LIN {X -195.246,Y +1107.046,Z +0.000,A -20.000,E1 +44.515,E3 +167624.420,E4 +0.000} C_DIS
LIN {X -198.051,Y +1092.368,Z +0.000,A -20.000,E1 +47.947,E3 +167640.946,E4 +0.000} C_DIS
LIN {X -198.143,Y +1081.370,Z +0.000,A -19.806,E1 +49.153,E3 +167652.807,E4 +0.000} C_DIS
LIN {X -197.177,Y +1073.569,Z +0.000,A -17.356,E1 +49.162,E3 +167661.391,E4 +0.000} C_DIS
LIN {X -195.448,Y +1066.139,Z +0.000,A -12.154,E1 +48.512,E3 +167669.986,E4 +0.000} C_DIS
LIN {X -193.346,Y +1058.941,Z +0.000,A -7.133,E1 +47.724,E3 +167678.866,E4 +0.000} C_DIS
LIN {X -191.781,Y +1050.839,Z +0.000,A -3.715,E1 +47.274,E3 +167689.199,E4 +0.000} C_DIS
LIN {X -190.795,Y +1039.355,Z +0.000,A -0.983,E1 +46.842,E3 +167703.859,E4 +0.000} C_DIS
LIN {X -190.395,Y +1028.856,Z +0.000,A -0.089,E1 +46.598,E3 +167717.253,E4 +0.000} C_DIS
LIN {X -190.239,Y +1018.851,Z +0.000,A -0.004,E1 +46.529,E3 +167730.021,E4 +0.000} C_DIS
LIN {X -190.161,Y +1004.975,Z +0.000,A +0.000,E1 +46.506,E3 +167747.735,E4 +0.000} C_DIS
LIN {X -190.142,Y +412.853,Z +0.000,A +0.000,E1 +46.501,E3 +168503.941,E4 +0.000} C_DIS
LIN {X -190.147,Y +401.077,Z +0.000,A +0.000,E1 +46.499,E3 +168518.982,E4 +0.000} C_DIS
LIN {X -190.159,Y +390.929,Z +0.000,A +0.000,E1 +46.494,E3 +168531.948,E4 +0.000} C_DIS
LIN {X -190.174,Y +383.973,Z +0.000,A +0.000,E1 +46.484,E3 +168540.841,E4 +0.000} C_DIS
LIN {X -190.200,Y +373.815,Z +0.000,A +0.000,E1 +46.448,E3 +168553.846,E4 +0.000} C_DIS
LIN {X -190.154,Y +361.003,Z +0.000,A +0.000,E1 +46.303,E3 +168570.340,E4 +0.000} C_DIS
LIN {X -189.772,Y +350.660,Z +0.000,A +0.049,E1 +45.996,E3 +168583.879,E4 +0.000} C_DIS
LIN {X -189.325,Y +346.917,Z +0.000,A +0.243,E1 +45.771,E3 +168588.948,E4 +0.000} C_DIS
LIN {X -188.196,Y +342.754,Z +0.000,A +1.966,E1 +45.249,E3 +168594.956,E4 +0.000} C_DIS
LIN {X -185.199,Y +337.023,Z +0.000,A +6.630,E1 +43.793,E3 +168604.330,E4 +0.000} C_DIS
LIN {X -181.141,Y +331.596,Z +0.000,A +12.274,E1 +41.569,E3 +168614.890,E4 +0.000} C_DIS
LIN {X -176.762,Y +326.804,Z +0.000,A +17.560,E1 +38.898,E3 +168626.314,E4 +0.000} C_DIS
LIN {X -172.184,Y +322.578,Z +0.000,A +19.859,E1 +36.197,E3 +168639.044,E4 +0.000} C_DIS
LIN {X -165.998,Y +317.874,Z +0.000,A +20.000,E1 +32.027,E3 +168658.802,E4 +0.000} C_DIS
LIN {X -160.137,Y +314.334,Z +0.000,A +20.000,E1 +26.368,E3 +168683.171,E4 +0.000} C_DIS
LIN {X -155.624,Y +312.245,Z +0.000,A +20.000,E1 +19.506,E3 +168711.847,E4 +0.000} C_DIS
LIN {X -153.557,Y +311.879,Z +0.000,A +20.000,E1 +11.113,E3 +168747.602,E4 +0.000} C_DIS
LIN {X -155.320,Y +313.348,Z +0.000,A +20.000,E1 +3.401,E3 +168780.786,E4 +0.000} C_DIS
LIN {X -160.005,Y +315.804,Z +0.000,A +20.000,E1 -4.720,E3 +168811.164,E4 +0.000} C_DIS
LIN {X -164.504,Y +318.255,Z +0.000,A +20.000,E1 -10.663,E3 +168830.533,E4 +0.000} C_DIS
LIN {X -170.340,Y +322.684,Z +0.000,A +20.000,E1 -17.457,E3 +168850.565,E4 +0.000} C_DIS
LIN {X -175.568,Y +329.106,Z +0.000,A +20.000,E1 -24.747,E3 +168867.799,E4 +0.000} C_DIS
LIN {X -184.074,Y +340.065,Z +0.000,A +20.000,E1 -33.664,E3 +168890.739,E4 +0.000} C_DIS
LIN {X -190.779,Y +351.388,Z +0.000,A +20.000,E1 -40.083,E3 +168908.517,E4 +0.000} C_DIS
LIN {X -195.254,Y +362.955,Z +0.000,A +20.000,E1 -44.515,E3 +168923.270,E4 +0.000} C_DIS
LIN {X -197.754,Y +374.780,Z +0.000,A +20.000,E1 -47.450,E3 +168936.692,E4 +0.000} C_DIS
LIN {X -198.310,Y +383.215,Z +0.000,A +19.956,E1 -48.698,E3 +168945.816,E4 +0.000} C_DIS
LIN {X -197.912,Y +391.275,Z +0.000,A +18.601,E1 -49.158,E3 +168954.534,E4 +0.000} C_DIS
LIN {X -196.679,Y +398.944,Z +0.000,A +13.989,E1 -48.784,E3 +168963.088,E4 +0.000} C_DIS
LIN {X -194.742,Y +406.288,Z +0.000,A +8.476,E1 -48.001,E3 +168971.771,E4 +0.000} C_DIS
LIN {X -192.748,Y +413.472,Z +0.000,A +3.905,E1 -47.267,E3 +168980.781,E4 +0.000} C_DIS
LIN {X -191.781,Y +419.162,Z +0.000,A +1.739,E1 -46.975,E3 +168988.049,E4 +0.000} C_DIS
LIN {X -190.795,Y +430.646,Z +0.000,A +0.152,E1 -46.707,E3 +169002.710,E4 +0.000} C_DIS
LIN {X -190.395,Y +441.145,Z +0.000,A +0.001,E1 -46.583,E3 +169016.103,E4 +0.000} C_DIS
LIN {X -190.239,Y +451.150,Z +0.000,A -0.000,E1 -46.528,E3 +169028.871,E4 +0.000} C_DIS
LIN {X -190.161,Y +465.026,Z +0.000,A -0.000,E1 -46.506,E3 +169046.586,E4 +0.000} C_DIS
LIN {X -190.142,Y +1057.148,Z +0.000,A -0.000,E1 -46.500,E3 +169802.792,E4 +0.000} C_DIS
LIN {X -190.147,Y +1068.924,Z +0.000,A -0.000,E1 -46.499,E3 +169817.833,E4 +0.000} C_DIS
LIN {X -190.159,Y +1079.072,Z +0.000,A -0.000,E1 -46.493,E3 +169830.798,E4 +0.000} C_DIS
LIN {X -190.174,Y +1086.028,Z +0.000,A -0.000,E1 -46.483,E3 +169839.692,E4 +0.000} C_DIS
LIN {X -190.200,Y +1096.186,Z +0.000,A -0.000,E1 -46.448,E3 +169852.696,E4 +0.000} C_DIS
LIN {X -190.154,Y +1108.998,Z +0.000,A -0.054,E1 -46.295,E3 +169869.191,E4 +0.000} C_DIS
LIN {X -189.772,Y +1119.341,Z +0.000,A -0.752,E1 -45.902,E3 +169882.729,E4 +0.000} C_DIS
LIN {X -189.097,Y +1124.276,Z +0.000,A -2.508,E1 -45.397,E3 +169889.461,E4 +0.000} C_DIS
LIN {X -187.410,Y +1129.069,Z +0.000,A -5.304,E1 -44.585,E3 +169896.634,E4 +0.000} C_DIS
LIN {X -183.899,Y +1134.873,Z +0.000,A -10.372,E1 -42.805,E3 +169906.640,E4 +0.000} C_DIS
LIN {X -179.711,Y +1140.065,Z +0.000,A -15.940,E1 -40.393,E3 +169917.426,E4 +0.000} C_DIS
LIN {X -176.763,Y +1143.197,Z +0.000,A -18.748,E1 -38.674,E3 +169925.164,E4 +0.000} C_DIS
LIN {X -172.185,Y +1147.423,Z +0.000,A -19.971,E1 -36.175,E3 +169937.894,E4 +0.000} C_DIS
LIN {X -165.999,Y +1152.127,Z +0.000,A -20.000,E1 -32.027,E3 +169957.652,E4 +0.000} C_DIS
LIN {X -160.138,Y +1155.667,Z +0.000,A -20.000,E1 -26.368,E3 +169982.022,E4 +0.000} C_DIS
LIN {X -155.625,Y +1157.756,Z +0.000,A -20.000,E1 -19.505,E3 +170010.698,E4 +0.000} C_DIS
LIN {X -153.552,Y +1158.113,Z +0.000,A -20.000,E1 -11.113,E3 +170046.449,E4 +0.000} C_DIS
LIN {X -156.311,Y +1155.540,Z +0.000,A -20.000,E1 -0.839,E3 +170089.809,E4 +0.000} C_DIS
LIN {X -161.281,Y +1151.851,Z +0.000,A -20.000,E1 +7.737,E3 +170119.708,E4 +0.000} C_DIS
LIN {X -167.493,Y +1147.157,Z +0.000,A -20.000,E1 +16.195,E3 +170144.147,E4 +0.000} C_DIS
LIN {X -173.235,Y +1142.221,Z +0.000,A -20.000,E1 +22.930,E3 +170161.449,E4 +0.000} C_DIS
LIN {X -181.123,Y +1133.734,Z +0.000,A -20.000,E1 +30.868,E3 +170182.205,E4 +0.000} C_DIS
LIN {X -189.654,Y +1120.856,Z +0.000,A -20.000,E1 +39.018,E3 +170204.219,E4 +0.000} C_DIS
LIN {X -195.246,Y +1107.046,Z +0.000,A -20.000,E1 +44.515,E3 +170222.121,E4 +0.000} C_DIS
LIN {X -198.051,Y +1092.368,Z +0.000,A -20.000,E1 +47.947,E3 +170238.647,E4 +0.000} C_DIS
LIN {X -198.143,Y +1081.370,Z +0.000,A -19.806,E1 +49.153,E3 +170250.508,E4 +0.000} C_DIS
LIN {X -197.177,Y +1073.569,Z +0.000,A -17.356,E1 +49.162,E3 +170259.092,E4 +0.000} C_DIS
LIN {X -195.448,Y +1066.139,Z +0.000,A -12.154,E1 +48.512,E3 +170267.687,E4 +0.000} C_DIS
LIN {X -193.346,Y +1058.941,Z +0.000,A -7.133,E1 +47.724,E3 +170276.567,E4 +0.000} C_DIS
LIN {X -191.781,Y +1050.839,Z +0.000,A -3.715,E1 +47.274,E3 +170286.900,E4 +0.000} C_DIS
LIN {X -190.795,Y +1039.355,Z +0.000,A -0.983,E1 +46.842,E3 +170301.560,E4 +0.000} C_DIS
LIN {X -190.395,Y +1028.856,Z +0.000,A -0.089,E1 +46.598,E3 +170314.954,E4 +0.000} C_DIS
LIN {X -190.239,Y +1018.851,Z +0.000,A -0.004,E1 +46.529,E3 +170327.722,E4 +0.000} C_DIS
LIN {X -190.161,Y +1004.975,Z +0.000,A +0.000,E1 +46.506,E3 +170345.436,E4 +0.000} C_DIS
LIN {X -190.142,Y +412.853,Z +0.000,A +0.000,E1 +46.501,E3 +171101.642,E4 +0.000} C_DIS
LIN {X -190.147,Y +401.077,Z +0.000,A +0.000,E1 +46.499,E3 +171116.683,E4 +0.000} C_DIS
LIN {X -190.159,Y +390.929,Z +0.000,A +0.000,E1 +46.494,E3 +171129.649,E4 +0.000} C_DIS
LIN {X -190.174,Y +383.973,Z +0.000,A +0.000,E1 +46.484,E3 +171138.542,E4 +0.000} C_DIS
LIN {X -190.200,Y +373.815,Z +0.000,A +0.000,E1 +46.448,E3 +171151.547,E4 +0.000} C_DIS
LIN {X -190.154,Y +361.003,Z +0.000,A +0.000,E1 +46.303,E3 +171168.041,E4 +0.000} C_DIS
LIN {X -189.772,Y +350.660,Z +0.000,A +0.049,E1 +45.996,E3 +171181.580,E4 +0.000} C_DIS
LIN {X -189.325,Y +346.917,Z +0.000,A +0.243,E1 +45.771,E3 +171186.649,E4 +0.000} C_DIS
LIN {X -188.196,Y +342.754,Z +0.000,A +1.966,E1 +45.249,E3 +171192.657,E4 +0.000} C_DIS
LIN {X -185.199,Y +337.023,Z +0.000,A +6.630,E1 +43.793,E3 +171202.031,E4 +0.000} C_DIS
LIN {X -181.141,Y +331.596,Z +0.000,A +12.274,E1 +41.569,E3 +171212.591,E4 +0.000} C_DIS
LIN {X -176.762,Y +326.804,Z +0.000,A +17.560,E1 +38.898,E3 +171224.015,E4 +0.000} C_DIS
LIN {X -172.184,Y +322.578,Z +0.000,A +19.859,E1 +36.197,E3 +171236.745,E4 +0.000} C_DIS
LIN {X -165.998,Y +317.874,Z +0.000,A +20.000,E1 +32.027,E3 +171256.503,E4 +0.000} C_DIS
LIN {X -160.137,Y +314.334,Z +0.000,A +20.000,E1 +26.368,E3 +171280.872,E4 +0.000} C_DIS
LIN {X -155.624,Y +312.245,Z +0.000,A +20.000,E1 +19.506,E3 +171309.548,E4 +0.000} C_DIS
LIN {X -153.557,Y +311.879,Z +0.000,A +20.000,E1 +11.113,E3 +171345.303,E4 +0.000} C_DIS
LIN {X -155.320,Y +313.348,Z +0.000,A +20.000,E1 +3.401,E3 +171378.487,E4 +0.000} C_DIS
LIN {X -160.005,Y +315.804,Z +0.000,A +20.000,E1 -4.720,E3 +171408.865,E4 +0.000} C_DIS
LIN {X -164.504,Y +318.255,Z +0.000,A +20.000,E1 -10.663,E3 +171428.234,E4 +0.000} C_DIS
LIN {X -170.340,Y +322.684,Z +0.000,A +20.000,E1 -17.457,E3 +171448.266,E4 +0.000} C_DIS
LIN {X -175.568,Y +329.106,Z +0.000,A +20.000,E1 -24.747,E3 +171465.500,E4 +0.000} C_DIS
LIN {X -184.074,Y +340.065,Z +0.000,A +20.000,E1 -33.664,E3 +171488.440,E4 +0.000} C_DIS
LIN {X -190.779,Y +351.388,Z +0.000,A +20.000,E1 -40.083,E3 +171506.218,E4 +0.000} C_DIS
LIN {X -195.254,Y +362.955,Z +0.000,A +20.000,E1 -44.515,E3 +171520.971,E4 +0.000} C_DIS
LIN {X -197.754,Y +374.780,Z +0.000,A +20.000,E1 -47.450,E3 +171534.393,E4 +0.000} C_DIS
LIN {X -198.310,Y +383.215,Z +0.000,A +19.956,E1 -48.698,E3 +171543.517,E4 +0.000} C_DIS
LIN {X -197.912,Y +391.275,Z +0.000,A +18.601,E1 -49.158,E3 +171552.235,E4 +0.000} C_DIS
LIN {X -196.679,Y +398.944,Z +0.000,A +13.989,E1 -48.784,E3 +171560.789,E4 +0.000} C_DIS
LIN {X -194.742,Y +406.288,Z +0.000,A +8.476,E1 -48.001,E3 +171569.472,E4 +0.000} C_DIS
LIN {X -192.748,Y +413.472,Z +0.000,A +3.905,E1 -47.267,E3 +171578.482,E4 +0.000} C_DIS
LIN {X -191.781,Y +419.162,Z +0.000,A +1.739,E1 -46.975,E3 +171585.750,E4 +0.000} C_DIS
LIN {X -190.795,Y +430.646,Z +0.000,A +0.152,E1 -46.707,E3 +171600.411,E4 +0.000} C_DIS
LIN {X -190.395,Y +441.145,Z +0.000,A +0.001,E1 -46.583,E3 +171613.804,E4 +0.000} C_DIS
LIN {X -190.239,Y +451.150,Z +0.000,A -0.000,E1 -46.528,E3 +171626.572,E4 +0.000} C_DIS
LIN {X -190.161,Y +465.026,Z +0.000,A -0.000,E1 -46.506,E3 +171644.287,E4 +0.000} C_DIS
LIN {X -190.142,Y +1057.148,Z +0.000,A -0.000,E1 -46.500,E3 +172400.493,E4 +0.000} C_DIS
LIN {X -190.147,Y +1068.924,Z +0.000,A -0.000,E1 -46.499,E3 +172415.534,E4 +0.000} C_DIS
LIN {X -190.159,Y +1079.072,Z +0.000,A -0.000,E1 -46.493,E3 +172428.499,E4 +0.000} C_DIS
LIN {X -190.174,Y +1086.028,Z +0.000,A -0.000,E1 -46.483,E3 +172437.393,E4 +0.000} C_DIS
LIN {X -190.200,Y +1096.186,Z +0.000,A -0.000,E1 -46.448,E3 +172450.397,E4 +0.000} C_DIS
LIN {X -190.154,Y +1108.998,Z +0.000,A -0.054,E1 -46.295,E3 +172466.892,E4 +0.000} C_DIS
LIN {X -189.772,Y +1119.341,Z +0.000,A -0.752,E1 -45.902,E3 +172480.430,E4 +0.000} C_DIS
LIN {X -189.097,Y +1124.276,Z +0.000,A -2.508,E1 -45.397,E3 +172487.162,E4 +0.000} C_DIS
LIN {X -187.410,Y +1129.069,Z +0.000,A -5.304,E1 -44.585,E3 +172494.335,E4 +0.000} C_DIS
LIN {X -183.899,Y +1134.873,Z +0.000,A -10.372,E1 -42.805,E3 +172504.341,E4 +0.000} C_DIS
LIN {X -179.711,Y +1140.065,Z +0.000,A -15.940,E1 -40.393,E3 +172515.127,E4 +0.000} C_DIS
LIN {X -176.763,Y +1143.197,Z +0.000,A -18.748,E1 -38.674,E3 +172522.865,E4 +0.000} C_DIS
LIN {X -172.185,Y +1147.423,Z +0.000,A -19.971,E1 -36.175,E3 +172535.595,E4 +0.000} C_DIS
LIN {X -165.999,Y +1152.127,Z +0.000,A -20.000,E1 -32.027,E3 +172555.353,E4 +0.000} C_DIS
LIN {X -160.138,Y +1155.667,Z +0.000,A -20.000,E1 -26.368,E3 +172579.723,E4 +0.000} C_DIS
LIN {X -155.625,Y +1157.756,Z +0.000,A -20.000,E1 -19.505,E3 +172608.399,E4 +0.000} C_DIS
LIN {X -153.552,Y +1158.113,Z +0.000,A -20.000,E1 -11.113,E3 +172644.150,E4 +0.000} C_DIS
LIN {X -156.311,Y +1155.540,Z +0.000,A -20.000,E1 -0.839,E3 +172687.510,E4 +0.000} C_DIS
LIN {X -161.281,Y +1151.851,Z +0.000,A -20.000,E1 +7.737,E3 +172717.409,E4 +0.000} C_DIS
LIN {X -167.493,Y +1147.157,Z +0.000,A -20.000,E1 +16.195,E3 +172741.848,E4 +0.000} C_DIS
LIN {X -173.235,Y +1142.221,Z +0.000,A -20.000,E1 +22.930,E3 +172759.150,E4 +0.000} C_DIS
LIN {X -181.123,Y +1133.734,Z +0.000,A -20.000,E1 +30.868,E3 +172779.906,E4 +0.000} C_DIS
LIN {X -189.654,Y +1120.856,Z +0.000,A -20.000,E1 +39.018,E3 +172801.920,E4 +0.000} C_DIS
LIN {X -195.246,Y +1107.046,Z +0.000,A -20.000,E1 +44.515,E3 +172819.822,E4 +0.000} C_DIS
LIN {X -198.051,Y +1092.368,Z +0.000,A -20.000,E1 +47.947,E3 +172836.348,E4 +0.000} C_DIS
LIN {X -198.143,Y +1081.370,Z +0.000,A -19.806,E1 +49.153,E3 +172848.209,E4 +0.000} C_DIS
LIN {X -197.177,Y +1073.569,Z +0.000,A -17.356,E1 +49.162,E3 +172856.793,E4 +0.000} C_DIS
LIN {X -195.448,Y +1066.139,Z +0.000,A -12.154,E1 +48.512,E3 +172865.388,E4 +0.000} C_DIS
LIN {X -193.346,Y +1058.941,Z +0.000,A -7.133,E1 +47.724,E3 +172874.268,E4 +0.000} C_DIS
LIN {X -191.781,Y +1050.839,Z +0.000,A -3.715,E1 +47.274,E3 +172884.601,E4 +0.000} C_DIS
LIN {X -190.795,Y +1039.355,Z +0.000,A -0.983,E1 +46.842,E3 +172899.261,E4 +0.000} C_DIS
LIN {X -190.395,Y +1028.856,Z +0.000,A -0.089,E1 +46.598,E3 +172912.655,E4 +0.000} C_DIS
LIN {X -190.239,Y +1018.851,Z +0.000,A -0.004,E1 +46.529,E3 +172925.423,E4 +0.000} C_DIS
LIN {X -190.161,Y +1004.975,Z +0.000,A +0.000,E1 +46.506,E3 +172943.137,E4 +0.000} C_DIS
LIN {X -190.142,Y +412.853,Z +0.000,A +0.000,E1 +46.501,E3 +173699.343,E4 +0.000} C_DIS
LIN {X -190.147,Y +401.077,Z +0.000,A +0.000,E1 +46.499,E3 +173714.384,E4 +0.000} C_DIS
LIN {X -190.159,Y +390.929,Z +0.000,A +0.000,E1 +46.494,E3 +173727.350,E4 +0.000} C_DIS
LIN {X -190.174,Y +383.973,Z +0.000,A +0.000,E1 +46.484,E3 +173736.243,E4 +0.000} C_DIS
LIN {X -190.200,Y +373.815,Z +0.000,A +0.000,E1 +46.448,E3 +173749.248,E4 +0.000} C_DIS
LIN {X -190.154,Y +361.003,Z +0.000,A +0.000,E1 +46.303,E3 +173765.742,E4 +0.000} C_DIS
LIN {X -189.772,Y +350.660,Z +0.000,A +0.049,E1 +45.996,E3 +173779.281,E4 +0.000} C_DIS
LIN {X -189.325,Y +346.917,Z +0.000,A +0.243,E1 +45.771,E3 +173784.350,E4 +0.000} C_DIS
LIN {X -188.196,Y +342.754,Z +0.000,A +1.966,E1 +45.249,E3 +173790.358,E4 +0.000} C_DIS
LIN {X -185.199,Y +337.023,Z +0.000,A +6.630,E1 +43.793,E3 +173799.732,E4 +0.000} C_DIS
LIN {X -181.141,Y +331.596,Z +0.000,A +12.274,E1 +41.569,E3 +173810.292,E4 +0.000} C_DIS
LIN {X -176.762,Y +326.804,Z +0.000,A +17.560,E1 +38.898,E3 +173821.716,E4 +0.000} C_DIS
LIN {X -172.184,Y +322.578,Z +0.000,A +19.859,E1 +36.197,E3 +173834.446,E4 +0.000} C_DIS
LIN {X -165.998,Y +317.874,Z +0.000,A +20.000,E1 +32.027,E3 +173854.204,E4 +0.000} C_DIS
LIN {X -160.137,Y +314.334,Z +0.000,A +20.000,E1 +26.368,E3 +173878.573,E4 +0.000} C_DIS
LIN {X -155.624,Y +312.245,Z +0.000,A +20.000,E1 +19.506,E3 +173907.249,E4 +0.000} C_DIS
LIN {X -153.557,Y +311.879,Z +0.000,A +20.000,E1 +11.113,E3 +173943.004,E4 +0.000} C_DIS
LIN {X -155.320,Y +313.348,Z +0.000,A +20.000,E1 +3.401,E3 +173976.188,E4 +0.000} C_DIS
LIN {X -160.005,Y +315.804,Z +0.000,A +20.000,E1 -4.720,E3 +174006.566,E4 +0.000} C_DIS
LIN {X -164.504,Y +318.255,Z +0.000,A +20.000,E1 -10.663,E3 +174025.935,E4 +0.000} C_DIS
LIN {X -170.340,Y +322.684,Z +0.000,A +20.000,E1 -17.457,E3 +174045.967,E4 +0.000} C_DIS
LIN {X -175.568,Y +329.106,Z +0.000,A +20.000,E1 -24.747,E3 +174063.201,E4 +0.000} C_DIS
LIN {X -184.074,Y +340.065,Z +0.000,A +20.000,E1 -33.664,E3 +174086.141,E4 +0.000} C_DIS
LIN {X -190.779,Y +351.388,Z +0.000,A +20.000,E1 -40.083,E3 +174103.919,E4 +0.000} C_DIS
LIN {X -195.254,Y +362.955,Z +0.000,A +20.000,E1 -44.515,E3 +174118.672,E4 +0.000} C_DIS
LIN {X -197.754,Y +374.780,Z +0.000,A +20.000,E1 -47.450,E3 +174132.094,E4 +0.000} C_DIS
LIN {X -198.310,Y +383.215,Z +0.000,A +19.956,E1 -48.698,E3 +174141.218,E4 +0.000} C_DIS
LIN {X -197.912,Y +391.275,Z +0.000,A +18.601,E1 -49.158,E3 +174149.936,E4 +0.000} C_DIS
LIN {X -196.679,Y +398.944,Z +0.000,A +13.989,E1 -48.784,E3 +174158.490,E4 +0.000} C_DIS
LIN {X -194.742,Y +406.288,Z +0.000,A +8.476,E1 -48.001,E3 +174167.173,E4 +0.000} C_DIS
LIN {X -192.748,Y +413.472,Z +0.000,A +3.905,E1 -47.267,E3 +174176.183,E4 +0.000} C_DIS
LIN {X -191.781,Y +419.162,Z +0.000,A +1.739,E1 -46.975,E3 +174183.451,E4 +0.000} C_DIS
LIN {X -190.795,Y +430.646,Z +0.000,A +0.152,E1 -46.707,E3 +174198.112,E4 +0.000} C_DIS
LIN {X -190.395,Y +441.145,Z +0.000,A +0.001,E1 -46.583,E3 +174211.505,E4 +0.000} C_DIS
LIN {X -190.239,Y +451.150,Z +0.000,A -0.000,E1 -46.528,E3 +174224.273,E4 +0.000} C_DIS
LIN {X -190.161,Y +465.026,Z +0.000,A -0.000,E1 -46.506,E3 +174241.988,E4 +0.000} C_DIS
LIN {X -190.142,Y +1057.148,Z +0.000,A -0.000,E1 -46.500,E3 +174998.194,E4 +0.000} C_DIS
LIN {X -190.147,Y +1068.924,Z +0.000,A -0.000,E1 -46.499,E3 +175013.235,E4 +0.000} C_DIS
LIN {X -190.159,Y +1079.072,Z +0.000,A -0.000,E1 -46.493,E3 +175026.200,E4 +0.000} C_DIS
LIN {X -190.174,Y +1086.028,Z +0.000,A -0.000,E1 -46.483,E3 +175035.094,E4 +0.000} C_DIS
LIN {X -190.200,Y +1096.186,Z +0.000,A -0.000,E1 -46.448,E3 +175048.098,E4 +0.000} C_DIS
LIN {X -190.154,Y +1108.998,Z +0.000,A -0.054,E1 -46.295,E3 +175064.593,E4 +0.000} C_DIS
LIN {X -189.772,Y +1119.341,Z +0.000,A -0.752,E1 -45.902,E3 +175078.131,E4 +0.000} C_DIS
LIN {X -189.097,Y +1124.276,Z +0.000,A -2.508,E1 -45.397,E3 +175084.863,E4 +0.000} C_DIS
LIN {X -187.410,Y +1129.069,Z +0.000,A -5.304,E1 -44.585,E3 +175092.036,E4 +0.000} C_DIS
LIN {X -183.899,Y +1134.873,Z +0.000,A -10.372,E1 -42.805,E3 +175102.042,E4 +0.000} C_DIS
LIN {X -179.711,Y +1140.065,Z +0.000,A -15.940,E1 -40.393,E3 +175112.828,E4 +0.000} C_DIS
LIN {X -176.763,Y +1143.197,Z +0.000,A -18.748,E1 -38.674,E3 +175120.566,E4 +0.000} C_DIS
LIN {X -172.185,Y +1147.423,Z +0.000,A -19.971,E1 -36.175,E3 +175133.296,E4 +0.000} C_DIS
LIN {X -165.999,Y +1152.127,Z +0.000,A -20.000,E1 -32.027,E3 +175153.054,E4 +0.000} C_DIS
LIN {X -160.138,Y +1155.667,Z +0.000,A -20.000,E1 -26.368,E3 +175177.424,E4 +0.000} C_DIS
LIN {X -155.625,Y +1157.756,Z +0.000,A -20.000,E1 -19.505,E3 +175206.100,E4 +0.000} C_DIS
LIN {X -153.552,Y +1158.113,Z +0.000,A -20.000,E1 -11.113,E3 +175241.851,E4 +0.000} C_DIS
LIN {X -156.311,Y +1155.540,Z +0.000,A -20.000,E1 -0.839,E3 +175285.211,E4 +0.000} C_DIS
LIN {X -161.281,Y +1151.851,Z +0.000,A -20.000,E1 +7.737,E3 +175315.110,E4 +0.000} C_DIS
LIN {X -167.493,Y +1147.157,Z +0.000,A -20.000,E1 +16.195,E3 +175339.549,E4 +0.000} C_DIS
LIN {X -173.235,Y +1142.221,Z +0.000,A -20.000,E1 +22.930,E3 +175356.851,E4 +0.000} C_DIS
LIN {X -181.123,Y +1133.734,Z +0.000,A -20.000,E1 +30.868,E3 +175377.607,E4 +0.000} C_DIS
LIN {X -189.654,Y +1120.856,Z +0.000,A -20.000,E1 +39.018,E3 +175399.621,E4 +0.000} C_DIS
LIN {X -195.246,Y +1107.046,Z +0.000,A -20.000,E1 +44.515,E3 +175417.523,E4 +0.000} C_DIS
LIN {X -198.051,Y +1092.368,Z +0.000,A -20.000,E1 +47.947,E3 +175434.049,E4 +0.000} C_DIS
LIN {X -198.143,Y +1081.370,Z +0.000,A -19.806,E1 +49.153,E3 +175445.910,E4 +0.000} C_DIS
LIN {X -197.177,Y +1073.569,Z +0.000,A -17.356,E1 +49.162,E3 +175454.494,E4 +0.000} C_DIS
LIN {X -195.448,Y +1066.139,Z +0.000,A -12.154,E1 +48.512,E3 +175463.089,E4 +0.000} C_DIS
LIN {X -193.346,Y +1058.941,Z +0.000,A -7.133,E1 +47.724,E3 +175471.969,E4 +0.000} C_DIS
LIN {X -191.781,Y +1050.839,Z +0.000,A -3.715,E1 +47.274,E3 +175482.302,E4 +0.000} C_DIS
LIN {X -190.795,Y +1039.355,Z +0.000,A -0.983,E1 +46.842,E3 +175496.962,E4 +0.000} C_DIS
LIN {X -190.395,Y +1028.856,Z +0.000,A -0.089,E1 +46.598,E3 +175510.356,E4 +0.000} C_DIS
LIN {X -190.239,Y +1018.851,Z +0.000,A -0.004,E1 +46.529,E3 +175523.124,E4 +0.000} C_DIS
LIN {X -190.161,Y +1004.975,Z +0.000,A +0.000,E1 +46.506,E3 +175540.838,E4 +0.000} C_DIS
LIN {X -190.142,Y +412.853,Z +0.000,A +0.000,E1 +46.501,E3 +176297.044,E4 +0.000} C_DIS
LIN {X -190.147,Y +401.077,Z +0.000,A +0.000,E1 +46.499,E3 +176312.085,E4 +0.000} C_DIS
LIN {X -190.159,Y +390.929,Z +0.000,A +0.000,E1 +46.494,E3 +176325.051,E4 +0.000} C_DIS
LIN {X -190.174,Y +383.973,Z +0.000,A +0.000,E1 +46.484,E3 +176333.944,E4 +0.000} C_DIS
LIN {X -190.200,Y +373.815,Z +0.000,A +0.000,E1 +46.448,E3 +176346.949,E4 +0.000} C_DIS
LIN {X -190.154,Y +361.003,Z +0.000,A +0.000,E1 +46.303,E3 +176363.443,E4 +0.000} C_DIS
LIN {X -189.772,Y +350.660,Z +0.000,A +0.049,E1 +45.996,E3 +176376.982,E4 +0.000} C_DIS
LIN {X -189.325,Y +346.917,Z +0.000,A +0.243,E1 +45.771,E3 +176382.051,E4 +0.000} C_DIS
LIN {X -188.196,Y +342.754,Z +0.000,A +1.966,E1 +45.249,E3 +176388.059,E4 +0.000} C_DIS
LIN {X -185.199,Y +337.023,Z +0.000,A +6.630,E1 +43.793,E3 +176397.433,E4 +0.000} C_DIS
LIN {X -181.141,Y +331.596,Z +0.000,A +12.274,E1 +41.569,E3 +176407.993,E4 +0.000} C_DIS
LIN {X -176.762,Y +326.804,Z +0.000,A +17.560,E1 +38.898,E3 +176419.417,E4 +0.000} C_DIS
LIN {X -172.184,Y +322.578,Z +0.000,A +19.859,E1 +36.197,E3 +176432.147,E4 +0.000} C_DIS
LIN {X -165.998,Y +317.874,Z +0.000,A +20.000,E1 +32.027,E3 +176451.905,E4 +0.000} C_DIS
LIN {X -160.137,Y +314.334,Z +0.000,A +20.000,E1 +26.368,E3 +176476.274,E4 +0.000} C_DIS
LIN {X -155.624,Y +312.245,Z +0.000,A +20.000,E1 +19.506,E3 +176504.950,E4 +0.000} C_DIS
LIN {X -153.557,Y +311.879,Z +0.000,A +20.000,E1 +11.113,E3 +176540.705,E4 +0.000} C_DIS
LIN {X -155.320,Y +313.348,Z +0.000,A +20.000,E1 +3.401,E3 +176573.889,E4 +0.000} C_DIS
LIN {X -160.005,Y +315.804,Z +0.000,A +20.000,E1 -4.720,E3 +176604.267,E4 +0.000} C_DIS
LIN {X -164.504,Y +318.255,Z +0.000,A +20.000,E1 -10.663,E3 +176623.636,E4 +0.000} C_DIS
LIN {X -170.340,Y +322.684,Z +0.000,A +20.000,E1 -17.457,E3 +176643.668,E4 +0.000} C_DIS
LIN {X -175.568,Y +329.106,Z +0.000,A +20.000,E1 -24.747,E3 +176660.902,E4 +0.000} C_DIS
LIN {X -184.074,Y +340.065,Z +0.000,A +20.000,E1 -33.664,E3 +176683.842,E4 +0.000} C_DIS
LIN {X -190.779,Y +351.388,Z +0.000,A +20.000,E1 -40.083,E3 +176701.620,E4 +0.000} C_DIS
LIN {X -195.254,Y +362.955,Z +0.000,A +20.000,E1 -44.515,E3 +176716.373,E4 +0.000} C_DIS
LIN {X -197.754,Y +374.780,Z +0.000,A +20.000,E1 -47.450,E3 +176729.795,E4 +0.000} C_DIS
LIN {X -198.310,Y +383.215,Z +0.000,A +19.956,E1 -48.698,E3 +176738.919,E4 +0.000} C_DIS
LIN {X -197.912,Y +391.275,Z +0.000,A +18.601,E1 -49.158,E3 +176747.637,E4 +0.000} C_DIS
LIN {X -196.679,Y +398.944,Z +0.000,A +13.989,E1 -48.784,E3 +176756.191,E4 +0.000} C_DIS
LIN {X -194.742,Y +406.288,Z +0.000,A +8.476,E1 -48.001,E3 +176764.874,E4 +0.000} C_DIS
LIN {X -192.748,Y +413.472,Z +0.000,A +3.905,E1 -47.267,E3 +176773.884,E4 +0.000} C_DIS
LIN {X -191.781,Y +419.162,Z +0.000,A +1.739,E1 -46.975,E3 +176781.152,E4 +0.000} C_DIS
LIN {X -190.795,Y +430.646,Z +0.000,A +0.152,E1 -46.707,E3 +176795.813,E4 +0.000} C_DIS
LIN {X -190.395,Y +441.145,Z +0.000,A +0.001,E1 -46.583,E3 +176809.206,E4 +0.000} C_DIS
LIN {X -190.239,Y +451.150,Z +0.000,A -0.000,E1 -46.528,E3 +176821.974,E4 +0.000} C_DIS
LIN {X -190.161,Y +465.026,Z +0.000,A -0.000,E1 -46.506,E3 +176839.689,E4 +0.000} C_DIS
LIN {X -190.142,Y +1057.148,Z +0.000,A -0.000,E1 -46.500,E3 +177595.895,E4 +0.000} C_DIS
LIN {X -190.147,Y +1068.924,Z +0.000,A -0.000,E1 -46.499,E3 +177610.936,E4 +0.000} C_DIS
LIN {X -190.159,Y +1079.072,Z +0.000,A -0.000,E1 -46.493,E3 +177623.901,E4 +0.000} C_DIS
LIN {X -190.174,Y +1086.028,Z +0.000,A -0.000,E1 -46.483,E3 +177632.795,E4 +0.000} C_DIS
LIN {X -190.200,Y +1096.186,Z +0.000,A -0.000,E1 -46.448,E3 +177645.799,E4 +0.000} C_DIS
LIN {X -190.154,Y +1108.998,Z +0.000,A -0.054,E1 -46.295,E3 +177662.294,E4 +0.000} C_DIS
LIN {X -189.772,Y +1119.341,Z +0.000,A -0.752,E1 -45.902,E3 +177675.832,E4 +0.000} C_DIS
LIN {X -189.097,Y +1124.276,Z +0.000,A -2.508,E1 -45.397,E3 +177682.564,E4 +0.000} C_DIS
LIN {X -187.410,Y +1129.069,Z +0.000,A -5.304,E1 -44.585,E3 +177689.737,E4 +0.000} C_DIS
LIN {X -183.899,Y +1134.873,Z +0.000,A -10.372,E1 -42.805,E3 +177699.743,E4 +0.000} C_DIS
LIN {X -179.711,Y +1140.065,Z +0.000,A -15.940,E1 -40.393,E3 +177710.529,E4 +0.000} C_DIS
LIN {X -176.763,Y +1143.197,Z +0.000,A -18.748,E1 -38.674,E3 +177718.267,E4 +0.000} C_DIS
LIN {X -172.185,Y +1147.423,Z +0.000,A -19.971,E1 -36.175,E3 +177730.997,E4 +0.000} C_DIS
LIN {X -165.999,Y +1152.127,Z +0.000,A -20.000,E1 -32.027,E3 +177750.755,E4 +0.000} C_DIS
LIN {X -160.138,Y +1155.667,Z +0.000,A -20.000,E1 -26.368,E3 +177775.125,E4 +0.000} C_DIS
LIN {X -155.625,Y +1157.756,Z +0.000,A -20.000,E1 -19.505,E3 +177803.801,E4 +0.000} C_DIS
LIN {X -153.552,Y +1158.113,Z +0.000,A -20.000,E1 -11.113,E3 +177839.552,E4 +0.000} C_DIS
LIN {X -156.311,Y +1155.540,Z +0.000,A -20.000,E1 -0.839,E3 +177882.912,E4 +0.000} C_DIS
LIN {X -161.281,Y +1151.851,Z +0.000,A -20.000,E1 +7.737,E3 +177912.811,E4 +0.000} C_DIS
LIN {X -167.493,Y +1147.157,Z +0.000,A -20.000,E1 +16.195,E3 +177937.250,E4 +0.000} C_DIS
LIN {X -173.235,Y +1142.221,Z +0.000,A -20.000,E1 +22.930,E3 +177954.552,E4 +0.000} C_DIS
LIN {X -181.123,Y +1133.734,Z +0.000,A -20.000,E1 +30.868,E3 +177975.308,E4 +0.000} C_DIS
LIN {X -189.654,Y +1120.856,Z +0.000,A -20.000,E1 +39.018,E3 +177997.322,E4 +0.000} C_DIS
LIN {X -195.246,Y +1107.046,Z +0.000,A -20.000,E1 +44.515,E3 +178015.224,E4 +0.000} C_DIS
LIN {X -198.051,Y +1092.368,Z +0.000,A -20.000,E1 +47.947,E3 +178031.750,E4 +0.000} C_DIS
LIN {X -198.143,Y +1081.370,Z +0.000,A -19.806,E1 +49.153,E3 +178043.611,E4 +0.000} C_DIS
LIN {X -197.177,Y +1073.569,Z +0.000,A -17.356,E1 +49.162,E3 +178052.195,E4 +0.000} C_DIS
LIN {X -195.448,Y +1066.139,Z +0.000,A -12.154,E1 +48.512,E3 +178060.790,E4 +0.000} C_DIS
LIN {X -193.346,Y +1058.941,Z +0.000,A -7.133,E1 +47.724,E3 +178069.670,E4 +0.000} C_DIS
LIN {X -191.781,Y +1050.839,Z +0.000,A -3.715,E1 +47.274,E3 +178080.003,E4 +0.000} C_DIS
LIN {X -190.795,Y +1039.355,Z +0.000,A -0.983,E1 +46.842,E3 +178094.663,E4 +0.000} C_DIS
LIN {X -190.395,Y +1028.856,Z +0.000,A -0.089,E1 +46.598,E3 +178108.057,E4 +0.000} C_DIS
LIN {X -190.239,Y +1018.851,Z +0.000,A -0.004,E1 +46.529,E3 +178120.825,E4 +0.000} C_DIS
LIN {X -190.161,Y +1004.975,Z +0.000,A +0.000,E1 +46.506,E3 +178138.539,E4 +0.000} C_DIS
LIN {X -190.142,Y +412.853,Z +0.000,A +0.000,E1 +46.501,E3 +178894.745,E4 +0.000} C_DIS
LIN {X -190.147,Y +401.077,Z +0.000,A +0.000,E1 +46.499,E3 +178909.786,E4 +0.000} C_DIS
LIN {X -190.159,Y +390.929,Z +0.000,A +0.000,E1 +46.494,E3 +178922.752,E4 +0.000} C_DIS
LIN {X -190.174,Y +383.973,Z +0.000,A +0.000,E1 +46.484,E3 +178931.645,E4 +0.000} C_DIS
LIN {X -190.200,Y +373.815,Z +0.000,A +0.000,E1 +46.448,E3 +178944.650,E4 +0.000} C_DIS
LIN {X -190.154,Y +361.003,Z +0.000,A +0.000,E1 +46.303,E3 +178961.144,E4 +0.000} C_DIS
LIN {X -189.772,Y +350.660,Z +0.000,A +0.049,E1 +45.996,E3 +178974.683,E4 +0.000} C_DIS
LIN {X -189.325,Y +346.917,Z +0.000,A +0.243,E1 +45.771,E3 +178979.752,E4 +0.000} C_DIS
LIN {X -188.196,Y +342.754,Z +0.000,A +1.966,E1 +45.249,E3 +178985.760,E4 +0.000} C_DIS
LIN {X -185.199,Y +337.023,Z +0.000,A +6.630,E1 +43.793,E3 +178995.134,E4 +0.000} C_DIS
LIN {X -181.141,Y +331.596,Z +0.000,A +12.274,E1 +41.569,E3 +179005.694,E4 +0.000} C_DIS
LIN {X -176.762,Y +326.804,Z +0.000,A +17.560,E1 +38.898,E3 +179017.118,E4 +0.000} C_DIS
LIN {X -172.184,Y +322.578,Z +0.000,A +19.859,E1 +36.197,E3 +179029.848,E4 +0.000} C_DIS
LIN {X -165.998,Y +317.874,Z +0.000,A +20.000,E1 +32.027,E3 +179049.606,E4 +0.000} C_DIS
LIN {X -160.137,Y +314.334,Z +0.000,A +20.000,E1 +26.368,E3 +179073.975,E4 +0.000} C_DIS
LIN {X -155.624,Y +312.245,Z +0.000,A +20.000,E1 +19.506,E3 +179102.651,E4 +0.000} C_DIS
LIN {X -153.557,Y +311.879,Z +0.000,A +20.000,E1 +11.113,E3 +179138.406,E4 +0.000} C_DIS
LIN {X -155.320,Y +313.348,Z +0.000,A +20.000,E1 +3.401,E3 +179171.590,E4 +0.000} C_DIS
LIN {X -160.005,Y +315.804,Z +0.000,A +20.000,E1 -4.720,E3 +179201.968,E4 +0.000} C_DIS
LIN {X -164.504,Y +318.255,Z +0.000,A +20.000,E1 -10.663,E3 +179221.337,E4 +0.000} C_DIS
LIN {X -170.340,Y +322.684,Z +0.000,A +20.000,E1 -17.457,E3 +179241.369,E4 +0.000} C_DIS
LIN {X -175.568,Y +329.106,Z +0.000,A +20.000,E1 -24.747,E3 +179258.603,E4 +0.000} C_DIS
LIN {X -184.074,Y +340.065,Z +0.000,A +20.000,E1 -33.664,E3 +179281.543,E4 +0.000} C_DIS
LIN {X -190.779,Y +351.388,Z +0.000,A +20.000,E1 -40.083,E3 +179299.321,E4 +0.000} C_DIS
LIN {X -195.254,Y +362.955,Z +0.000,A +20.000,E1 -44.515,E3 +179314.074,E4 +0.000} C_DIS
LIN {X -197.754,Y +374.780,Z +0.000,A +20.000,E1 -47.450,E3 +179327.496,E4 +0.000} C_DIS
LIN {X -198.310,Y +383.215,Z +0.000,A +19.956,E1 -48.698,E3 +179336.620,E4 +0.000} C_DIS
LIN {X -197.912,Y +391.275,Z +0.000,A +18.601,E1 -49.158,E3 +179345.338,E4 +0.000} C_DIS
LIN {X -196.679,Y +398.944,Z +0.000,A +13.989,E1 -48.784,E3 +179353.892,E4 +0.000} C_DIS
LIN {X -194.742,Y +406.288,Z +0.000,A +8.476,E1 -48.001,E3 +179362.575,E4 +0.000} C_DIS
LIN {X -192.748,Y +413.472,Z +0.000,A +3.905,E1 -47.267,E3 +179371.585,E4 +0.000} C_DIS
LIN {X -191.781,Y +419.162,Z +0.000,A +1.739,E1 -46.975,E3 +179378.853,E4 +0.000} C_DIS
LIN {X -190.795,Y +430.646,Z +0.000,A +0.152,E1 -46.707,E3 +179393.514,E4 +0.000} C_DIS
LIN {X -190.395,Y +441.145,Z +0.000,A +0.001,E1 -46.583,E3 +179406.907,E4 +0.000} C_DIS
LIN {X -190.239,Y +451.150,Z +0.000,A -0.000,E1 -46.528,E3 +179419.675,E4 +0.000} C_DIS
LIN {X -190.161,Y +465.026,Z +0.000,A -0.000,E1 -46.506,E3 +179437.390,E4 +0.000} C_DIS
LIN {X -190.142,Y +1057.148,Z +0.000,A -0.000,E1 -46.500,E3 +180193.596,E4 +0.000} C_DIS
LIN {X -190.147,Y +1068.924,Z +0.000,A -0.000,E1 -46.499,E3 +180208.637,E4 +0.000} C_DIS
LIN {X -190.159,Y +1079.072,Z +0.000,A -0.000,E1 -46.493,E3 +180221.602,E4 +0.000} C_DIS
LIN {X -190.174,Y +1086.028,Z +0.000,A -0.000,E1 -46.483,E3 +180230.496,E4 +0.000} C_DIS
LIN {X -190.200,Y +1096.186,Z +0.000,A -0.000,E1 -46.448,E3 +180243.500,E4 +0.000} C_DIS
LIN {X -190.154,Y +1108.998,Z +0.000,A -0.054,E1 -46.295,E3 +180259.995,E4 +0.000} C_DIS
LIN {X -189.772,Y +1119.341,Z +0.000,A -0.752,E1 -45.902,E3 +180273.533,E4 +0.000} C_DIS
LIN {X -189.097,Y +1124.276,Z +0.000,A -2.508,E1 -45.397,E3 +180280.265,E4 +0.000} C_DIS
LIN {X -187.410,Y +1129.069,Z +0.000,A -5.304,E1 -44.585,E3 +180287.438,E4 +0.000} C_DIS
LIN {X -183.899,Y +1134.873,Z +0.000,A -10.372,E1 -42.805,E3 +180297.444,E4 +0.000} C_DIS
LIN {X -179.711,Y +1140.065,Z +0.000,A -15.940,E1 -40.393,E3 +180308.230,E4 +0.000} C_DIS
LIN {X -176.763,Y +1143.197,Z +0.000,A -18.748,E1 -38.674,E3 +180315.968,E4 +0.000} C_DIS
LIN {X -172.185,Y +1147.423,Z +0.000,A -19.971,E1 -36.175,E3 +180328.698,E4 +0.000} C_DIS
LIN {X -165.999,Y +1152.127,Z +0.000,A -20.000,E1 -32.027,E3 +180348.456,E4 +0.000} C_DIS
LIN {X -160.138,Y +1155.667,Z +0.000,A -20.000,E1 -26.368,E3 +180372.826,E4 +0.000} C_DIS
LIN {X -155.625,Y +1157.756,Z +0.000,A -20.000,E1 -19.505,E3 +180401.502,E4 +0.000} C_DIS
LIN {X -153.552,Y +1158.113,Z +0.000,A -20.000,E1 -11.113,E3 +180437.253,E4 +0.000} C_DIS
LIN {X -156.311,Y +1155.540,Z +0.000,A -20.000,E1 -0.839,E3 +180480.613,E4 +0.000} C_DIS
LIN {X -161.281,Y +1151.851,Z +0.000,A -20.000,E1 +7.737,E3 +180510.512,E4 +0.000} C_DIS
LIN {X -167.493,Y +1147.157,Z +0.000,A -20.000,E1 +16.195,E3 +180534.951,E4 +0.000} C_DIS
LIN {X -173.235,Y +1142.221,Z +0.000,A -20.000,E1 +22.930,E3 +180552.253,E4 +0.000} C_DIS
LIN {X -181.123,Y +1133.734,Z +0.000,A -20.000,E1 +30.868,E3 +180573.009,E4 +0.000} C_DIS
LIN {X -189.654,Y +1120.856,Z +0.000,A -20.000,E1 +39.018,E3 +180595.023,E4 +0.000} C_DIS
LIN {X -195.246,Y +1107.046,Z +0.000,A -20.000,E1 +44.515,E3 +180612.925,E4 +0.000} C_DIS
LIN {X -198.051,Y +1092.368,Z +0.000,A -20.000,E1 +47.947,E3 +180629.451,E4 +0.000} C_DIS
LIN {X -198.143,Y +1081.370,Z +0.000,A -19.806,E1 +49.153,E3 +180641.312,E4 +0.000} C_DIS
LIN {X -197.177,Y +1073.569,Z +0.000,A -17.356,E1 +49.162,E3 +180649.896,E4 +0.000} C_DIS
LIN {X -195.448,Y +1066.139,Z +0.000,A -12.154,E1 +48.512,E3 +180658.491,E4 +0.000} C_DIS
LIN {X -193.346,Y +1058.941,Z +0.000,A -7.133,E1 +47.724,E3 +180667.371,E4 +0.000} C_DIS
LIN {X -191.781,Y +1050.839,Z +0.000,A -3.715,E1 +47.274,E3 +180677.704,E4 +0.000} C_DIS
LIN {X -190.795,Y +1039.355,Z +0.000,A -0.983,E1 +46.842,E3 +180692.364,E4 +0.000} C_DIS
LIN {X -190.395,Y +1028.856,Z +0.000,A -0.089,E1 +46.598,E3 +180705.758,E4 +0.000} C_DIS
LIN {X -190.239,Y +1018.851,Z +0.000,A -0.004,E1 +46.529,E3 +180718.526,E4 +0.000} C_DIS
LIN {X -190.161,Y +1004.975,Z +0.000,A +0.000,E1 +46.506,E3 +180736.240,E4 +0.000} C_DIS
LIN {X -190.142,Y +412.853,Z +0.000,A +0.000,E1 +46.501,E3 +181492.446,E4 +0.000} C_DIS
LIN {X -190.147,Y +401.077,Z +0.000,A +0.000,E1 +46.499,E3 +181507.487,E4 +0.000} C_DIS
LIN {X -190.159,Y +390.929,Z +0.000,A +0.000,E1 +46.494,E3 +181520.453,E4 +0.000} C_DIS
LIN {X -190.174,Y +383.973,Z +0.000,A +0.000,E1 +46.484,E3 +181529.346,E4 +0.000} C_DIS
LIN {X -190.200,Y +373.815,Z +0.000,A +0.000,E1 +46.448,E3 +181542.351,E4 +0.000} C_DIS
LIN {X -190.154,Y +361.003,Z +0.000,A +0.000,E1 +46.303,E3 +181558.845,E4 +0.000} C_DIS
LIN {X -189.772,Y +350.660,Z +0.000,A +0.049,E1 +45.996,E3 +181572.384,E4 +0.000} C_DIS
LIN {X -189.325,Y +346.917,Z +0.000,A +0.243,E1 +45.771,E3 +181577.453,E4 +0.000} C_DIS
LIN {X -188.196,Y +342.754,Z +0.000,A +1.966,E1 +45.249,E3 +181583.461,E4 +0.000} C_DIS
LIN {X -185.199,Y +337.023,Z +0.000,A +6.630,E1 +43.793,E3 +181592.835,E4 +0.000} C_DIS
LIN {X -181.141,Y +331.596,Z +0.000,A +12.274,E1 +41.569,E3 +181603.395,E4 +0.000} C_DIS
LIN {X -176.762,Y +326.804,Z +0.000,A +17.560,E1 +38.898,E3 +181614.819,E4 +0.000} C_DIS
LIN {X -172.184,Y +322.578,Z +0.000,A +19.859,E1 +36.197,E3 +181627.549,E4 +0.000} C_DIS
LIN {X -165.998,Y +317.874,Z +0.000,A +20.000,E1 +32.027,E3 +181647.307,E4 +0.000} C_DIS
LIN {X -160.137,Y +314.334,Z +0.000,A +20.000,E1 +26.368,E3 +181671.676,E4 +0.000} C_DIS
LIN {X -155.624,Y +312.245,Z +0.000,A +20.000,E1 +19.506,E3 +181700.352,E4 +0.000} C_DIS
LIN {X -153.557,Y +311.879,Z +0.000,A +20.000,E1 +11.113,E3 +181736.107,E4 +0.000} C_DIS
LIN {X -155.320,Y +313.348,Z +0.000,A +20.000,E1 +3.401,E3 +181769.291,E4 +0.000} C_DIS
LIN {X -160.005,Y +315.804,Z +0.000,A +20.000,E1 -4.720,E3 +181799.669,E4 +0.000} C_DIS
LIN {X -164.504,Y +318.255,Z +0.000,A +20.000,E1 -10.663,E3 +181819.038,E4 +0.000} C_DIS
LIN {X -170.340,Y +322.684,Z +0.000,A +20.000,E1 -17.457,E3 +181839.070,E4 +0.000} C_DIS
LIN {X -175.568,Y +329.106,Z +0.000,A +20.000,E1 -24.747,E3 +181856.304,E4 +0.000} C_DIS
LIN {X -184.074,Y +340.065,Z +0.000,A +20.000,E1 -33.664,E3 +181879.244,E4 +0.000} C_DIS
LIN {X -190.779,Y +351.388,Z +0.000,A +20.000,E1 -40.083,E3 +181897.022,E4 +0.000} C_DIS
LIN {X -195.254,Y +362.955,Z +0.000,A +20.000,E1 -44.515,E3 +181911.775,E4 +0.000} C_DIS
LIN {X -197.754,Y +374.780,Z +0.000,A +20.000,E1 -47.450,E3 +181925.197,E4 +0.000} C_DIS
LIN {X -198.310,Y +383.215,Z +0.000,A +19.956,E1 -48.698,E3 +181934.321,E4 +0.000} C_DIS
LIN {X -197.912,Y +391.275,Z +0.000,A +18.601,E1 -49.158,E3 +181943.039,E4 +0.000} C_DIS
LIN {X -196.679,Y +398.944,Z +0.000,A +13.989,E1 -48.784,E3 +181951.593,E4 +0.000} C_DIS
LIN {X -194.742,Y +406.288,Z +0.000,A +8.476,E1 -48.001,E3 +181960.276,E4 +0.000} C_DIS
LIN {X -192.748,Y +413.472,Z +0.000,A +3.905,E1 -47.267,E3 +181969.286,E4 +0.000} C_DIS
LIN {X -191.781,Y +419.162,Z +0.000,A +1.739,E1 -46.975,E3 +181976.554,E4 +0.000} C_DIS
LIN {X -190.795,Y +430.646,Z +0.000,A +0.152,E1 -46.707,E3 +181991.215,E4 +0.000} C_DIS
LIN {X -190.395,Y +441.145,Z +0.000,A +0.001,E1 -46.583,E3 +182004.608,E4 +0.000} C_DIS
LIN {X -190.239,Y +451.150,Z +0.000,A -0.000,E1 -46.528,E3 +182017.376,E4 +0.000} C_DIS
LIN {X -190.161,Y +465.026,Z +0.000,A -0.000,E1 -46.506,E3 +182035.091,E4 +0.000} C_DIS
LIN {X -190.142,Y +1057.148,Z +0.000,A -0.000,E1 -46.500,E3 +182791.297,E4 +0.000} C_DIS
LIN {X -190.147,Y +1068.924,Z +0.000,A -0.000,E1 -46.499,E3 +182806.338,E4 +0.000} C_DIS
LIN {X -190.159,Y +1079.072,Z +0.000,A -0.000,E1 -46.493,E3 +182819.303,E4 +0.000} C_DIS
LIN {X -190.174,Y +1086.028,Z +0.000,A -0.000,E1 -46.483,E3 +182828.197,E4 +0.000} C_DIS
LIN {X -190.200,Y +1096.186,Z +0.000,A -0.000,E1 -46.448,E3 +182841.201,E4 +0.000} C_DIS
LIN {X -190.154,Y +1108.998,Z +0.000,A -0.054,E1 -46.295,E3 +182857.696,E4 +0.000} C_DIS
LIN {X -189.772,Y +1119.341,Z +0.000,A -0.752,E1 -45.902,E3 +182871.234,E4 +0.000} C_DIS
LIN {X -189.097,Y +1124.276,Z +0.000,A -2.508,E1 -45.397,E3 +182877.966,E4 +0.000} C_DIS
LIN {X -187.410,Y +1129.069,Z +0.000,A -5.304,E1 -44.585,E3 +182885.139,E4 +0.000} C_DIS
LIN {X -183.899,Y +1134.873,Z +0.000,A -10.372,E1 -42.805,E3 +182895.145,E4 +0.000} C_DIS
LIN {X -179.711,Y +1140.065,Z +0.000,A -15.940,E1 -40.393,E3 +182905.931,E4 +0.000} C_DIS
LIN {X -176.763,Y +1143.197,Z +0.000,A -18.748,E1 -38.674,E3 +182913.669,E4 +0.000} C_DIS
LIN {X -172.185,Y +1147.423,Z +0.000,A -19.971,E1 -36.175,E3 +182926.399,E4 +0.000} C_DIS
LIN {X -165.999,Y +1152.127,Z +0.000,A -20.000,E1 -32.027,E3 +182946.157,E4 +0.000} C_DIS
LIN {X -160.138,Y +1155.667,Z +0.000,A -20.000,E1 -26.368,E3 +182970.527,E4 +0.000} C_DIS
LIN {X -155.625,Y +1157.756,Z +0.000,A -20.000,E1 -19.505,E3 +182999.203,E4 +0.000} C_DIS
LIN {X -153.552,Y +1158.113,Z +0.000,A -20.000,E1 -11.113,E3 +183034.954,E4 +0.000} C_DIS
LIN {X -156.311,Y +1155.540,Z +0.000,A -20.000,E1 -0.839,E3 +183078.314,E4 +0.000} C_DIS
LIN {X -161.281,Y +1151.851,Z +0.000,A -20.000,E1 +7.737,E3 +183108.213,E4 +0.000} C_DIS
LIN {X -167.493,Y +1147.157,Z +0.000,A -20.000,E1 +16.195,E3 +183132.652,E4 +0.000} C_DIS
LIN {X -173.235,Y +1142.221,Z +0.000,A -20.000,E1 +22.930,E3 +183149.954,E4 +0.000} C_DIS
LIN {X -181.123,Y +1133.734,Z +0.000,A -20.000,E1 +30.868,E3 +183170.710,E4 +0.000} C_DIS
LIN {X -189.654,Y +1120.856,Z +0.000,A -20.000,E1 +39.018,E3 +183192.724,E4 +0.000} C_DIS
LIN {X -195.246,Y +1107.046,Z +0.000,A -20.000,E1 +44.515,E3 +183210.626,E4 +0.000} C_DIS
LIN {X -198.051,Y +1092.368,Z +0.000,A -20.000,E1 +47.947,E3 +183227.152,E4 +0.000} C_DIS
LIN {X -198.143,Y +1081.370,Z +0.000,A -19.806,E1 +49.153,E3 +183239.013,E4 +0.000} C_DIS
LIN {X -197.177,Y +1073.569,Z +0.000,A -17.356,E1 +49.162,E3 +183247.597,E4 +0.000} C_DIS
LIN {X -195.448,Y +1066.139,Z +0.000,A -12.154,E1 +48.512,E3 +183256.192,E4 +0.000} C_DIS
LIN {X -193.346,Y +1058.941,Z +0.000,A -7.133,E1 +47.724,E3 +183265.072,E4 +0.000} C_DIS
LIN {X -191.781,Y +1050.839,Z +0.000,A -3.715,E1 +47.274,E3 +183275.405,E4 +0.000} C_DIS
LIN {X -190.795,Y +1039.355,Z +0.000,A -0.983,E1 +46.842,E3 +183290.065,E4 +0.000} C_DIS
LIN {X -190.395,Y +1028.856,Z +0.000,A -0.089,E1 +46.598,E3 +183303.459,E4 +0.000} C_DIS
LIN {X -190.239,Y +1018.851,Z +0.000,A -0.004,E1 +46.529,E3 +183316.227,E4 +0.000} C_DIS
LIN {X -190.161,Y +1004.975,Z +0.000,A +0.000,E1 +46.506,E3 +183333.941,E4 +0.000} C_DIS
LIN {X -190.142,Y +412.853,Z +0.000,A +0.000,E1 +46.501,E3 +184090.147,E4 +0.000} C_DIS
LIN {X -190.147,Y +401.077,Z +0.000,A +0.000,E1 +46.499,E3 +184105.188,E4 +0.000} C_DIS
LIN {X -190.159,Y +390.929,Z +0.000,A +0.000,E1 +46.494,E3 +184118.154,E4 +0.000} C_DIS
LIN {X -190.174,Y +383.973,Z +0.000,A +0.000,E1 +46.484,E3 +184127.047,E4 +0.000} C_DIS
LIN {X -190.200,Y +373.815,Z +0.000,A +0.000,E1 +46.448,E3 +184140.052,E4 +0.000} C_DIS
LIN {X -190.154,Y +361.003,Z +0.000,A +0.000,E1 +46.303,E3 +184156.546,E4 +0.000} C_DIS
LIN {X -189.772,Y +350.660,Z +0.000,A +0.049,E1 +45.996,E3 +184170.085,E4 +0.000} C_DIS
LIN {X -189.325,Y +346.917,Z +0.000,A +0.243,E1 +45.771,E3 +184175.154,E4 +0.000} C_DIS
LIN {X -188.196,Y +342.754,Z +0.000,A +1.966,E1 +45.249,E3 +184181.162,E4 +0.000} C_DIS
LIN {X -185.199,Y +337.023,Z +0.000,A +6.630,E1 +43.793,E3 +184190.536,E4 +0.000} C_DIS
LIN {X -181.141,Y +331.596,Z +0.000,A +12.274,E1 +41.569,E3 +184201.096,E4 +0.000} C_DIS
LIN {X -176.762,Y +326.804,Z +0.000,A +17.560,E1 +38.898,E3 +184212.520,E4 +0.000} C_DIS
LIN {X -172.184,Y +322.578,Z +0.000,A +19.859,E1 +36.197,E3 +184225.250,E4 +0.000} C_DIS
LIN {X -165.998,Y +317.874,Z +0.000,A +20.000,E1 +32.027,E3 +184245.008,E4 +0.000} C_DIS
LIN {X -160.137,Y +314.334,Z +0.000,A +20.000,E1 +26.368,E3 +184269.377,E4 +0.000} C_DIS
LIN {X -155.624,Y +312.245,Z +0.000,A +20.000,E1 +19.506,E3 +184298.053,E4 +0.000} C_DIS
LIN {X -153.557,Y +311.879,Z +0.000,A +20.000,E1 +11.113,E3 +184333.808,E4 +0.000} C_DIS
LIN {X -155.320,Y +313.348,Z +0.000,A +20.000,E1 +3.401,E3 +184366.992,E4 +0.000} C_DIS
LIN {X -160.005,Y +315.804,Z +0.000,A +20.000,E1 -4.720,E3 +184397.370,E4 +0.000} C_DIS
LIN {X -164.504,Y +318.255,Z +0.000,A +20.000,E1 -10.663,E3 +184416.739,E4 +0.000} C_DIS
LIN {X -170.340,Y +322.684,Z +0.000,A +20.000,E1 -17.457,E3 +184436.771,E4 +0.000} C_DIS
LIN {X -175.568,Y +329.106,Z +0.000,A +20.000,E1 -24.747,E3 +184454.005,E4 +0.000} C_DIS
LIN {X -184.074,Y +340.065,Z +0.000,A +20.000,E1 -33.664,E3 +184476.945,E4 +0.000} C_DIS
LIN {X -190.779,Y +351.388,Z +0.000,A +20.000,E1 -40.083,E3 +184494.723,E4 +0.000} C_DIS
LIN {X -195.254,Y +362.955,Z +0.000,A +20.000,E1 -44.515,E3 +184509.476,E4 +0.000} C_DIS
LIN {X -197.754,Y +374.780,Z +0.000,A +20.000,E1 -47.450,E3 +184522.898,E4 +0.000} C_DIS
LIN {X -198.310,Y +383.215,Z +0.000,A +19.956,E1 -48.698,E3 +184532.022,E4 +0.000} C_DIS
LIN {X -197.912,Y +391.275,Z +0.000,A +18.601,E1 -49.158,E3 +184540.740,E4 +0.000} C_DIS
LIN {X -196.679,Y +398.944,Z +0.000,A +13.989,E1 -48.784,E3 +184549.294,E4 +0.000} C_DIS
LIN {X -194.742,Y +406.288,Z +0.000,A +8.476,E1 -48.001,E3 +184557.977,E4 +0.000} C_DIS
LIN {X -192.748,Y +413.472,Z +0.000,A +3.905,E1 -47.267,E3 +184566.987,E4 +0.000} C_DIS
LIN {X -191.781,Y +419.162,Z +0.000,A +1.739,E1 -46.975,E3 +184574.255,E4 +0.000} C_DIS
LIN {X -190.795,Y +430.646,Z +0.000,A +0.152,E1 -46.707,E3 +184588.916,E4 +0.000} C_DIS
LIN {X -190.395,Y +441.145,Z +0.000,A +0.001,E1 -46.583,E3 +184602.309,E4 +0.000} C_DIS
LIN {X -190.239,Y +451.150,Z +0.000,A -0.000,E1 -46.528,E3 +184615.077,E4 +0.000} C_DIS
LIN {X -190.161,Y +465.026,Z +0.000,A -0.000,E1 -46.506,E3 +184632.792,E4 +0.000} C_DIS
LIN {X -190.142,Y +1057.148,Z +0.000,A -0.000,E1 -46.500,E3 +185388.998,E4 +0.000} C_DIS
LIN {X -190.147,Y +1068.924,Z +0.000,A -0.000,E1 -46.499,E3 +185404.039,E4 +0.000} C_DIS
LIN {X -190.159,Y +1079.072,Z +0.000,A -0.000,E1 -46.493,E3 +185417.004,E4 +0.000} C_DIS
LIN {X -190.174,Y +1086.028,Z +0.000,A -0.000,E1 -46.483,E3 +185425.898,E4 +0.000} C_DIS
LIN {X -190.200,Y +1096.186,Z +0.000,A -0.000,E1 -46.448,E3 +185438.902,E4 +0.000} C_DIS
LIN {X -190.154,Y +1108.998,Z +0.000,A -0.054,E1 -46.295,E3 +185455.397,E4 +0.000} C_DIS
LIN {X -189.772,Y +1119.341,Z +0.000,A -0.752,E1 -45.902,E3 +185468.935,E4 +0.000} C_DIS
LIN {X -189.097,Y +1124.276,Z +0.000,A -2.508,E1 -45.397,E3 +185475.667,E4 +0.000} C_DIS
LIN {X -187.410,Y +1129.069,Z +0.000,A -5.304,E1 -44.585,E3 +185482.840,E4 +0.000} C_DIS
LIN {X -183.899,Y +1134.873,Z +0.000,A -10.372,E1 -42.805,E3 +185492.846,E4 +0.000} C_DIS
LIN {X -179.711,Y +1140.065,Z +0.000,A -15.940,E1 -40.393,E3 +185503.632,E4 +0.000} C_DIS
LIN {X -176.763,Y +1143.197,Z +0.000,A -18.748,E1 -38.674,E3 +185511.370,E4 +0.000} C_DIS
LIN {X -172.185,Y +1147.423,Z +0.000,A -19.971,E1 -36.175,E3 +185524.100,E4 +0.000} C_DIS
LIN {X -165.999,Y +1152.127,Z +0.000,A -20.000,E1 -32.027,E3 +185543.858,E4 +0.000} C_DIS
LIN {X -160.138,Y +1155.667,Z +0.000,A -20.000,E1 -26.368,E3 +185568.228,E4 +0.000} C_DIS
LIN {X -155.625,Y +1157.756,Z +0.000,A -20.000,E1 -19.505,E3 +185596.904,E4 +0.000} C_DIS
LIN {X -153.552,Y +1158.113,Z +0.000,A -20.000,E1 -11.113,E3 +185632.655,E4 +0.000} C_DIS
LIN {X -156.311,Y +1155.540,Z +0.000,A -20.000,E1 -0.839,E3 +185676.015,E4 +0.000} C_DIS
LIN {X -161.281,Y +1151.851,Z +0.000,A -20.000,E1 +7.737,E3 +185705.914,E4 +0.000} C_DIS
LIN {X -167.493,Y +1147.157,Z +0.000,A -20.000,E1 +16.195,E3 +185730.353,E4 +0.000} C_DIS
LIN {X -173.235,Y +1142.221,Z +0.000,A -20.000,E1 +22.930,E3 +185747.655,E4 +0.000} C_DIS
LIN {X -181.123,Y +1133.734,Z +0.000,A -20.000,E1 +30.868,E3 +185768.411,E4 +0.000} C_DIS
LIN {X -189.654,Y +1120.856,Z +0.000,A -20.000,E1 +39.018,E3 +185790.425,E4 +0.000} C_DIS
LIN {X -195.246,Y +1107.046,Z +0.000,A -20.000,E1 +44.515,E3 +185808.327,E4 +0.000} C_DIS
LIN {X -198.051,Y +1092.368,Z +0.000,A -20.000,E1 +47.947,E3 +185824.853,E4 +0.000} C_DIS
LIN {X -198.143,Y +1081.370,Z +0.000,A -19.806,E1 +49.153,E3 +185836.714,E4 +0.000} C_DIS
LIN {X -197.177,Y +1073.569,Z +0.000,A -17.356,E1 +49.162,E3 +185845.298,E4 +0.000} C_DIS
LIN {X -195.448,Y +1066.139,Z +0.000,A -12.154,E1 +48.512,E3 +185853.893,E4 +0.000} C_DIS
LIN {X -193.346,Y +1058.941,Z +0.000,A -7.133,E1 +47.724,E3 +185862.773,E4 +0.000} C_DIS
LIN {X -191.781,Y +1050.839,Z +0.000,A -3.715,E1 +47.274,E3 +185873.106,E4 +0.000} C_DIS
LIN {X -190.795,Y +1039.355,Z +0.000,A -0.983,E1 +46.842,E3 +185887.766,E4 +0.000} C_DIS
LIN {X -190.395,Y +1028.856,Z +0.000,A -0.089,E1 +46.598,E3 +185901.160,E4 +0.000} C_DIS
LIN {X -190.239,Y +1018.851,Z +0.000,A -0.004,E1 +46.529,E3 +185913.928,E4 +0.000} C_DIS
LIN {X -190.161,Y +1004.975,Z +0.000,A +0.000,E1 +46.506,E3 +185931.642,E4 +0.000} C_DIS
LIN {X -190.142,Y +412.853,Z +0.000,A +0.000,E1 +46.501,E3 +186687.848,E4 +0.000} C_DIS
LIN {X -190.147,Y +401.077,Z +0.000,A +0.000,E1 +46.499,E3 +186702.889,E4 +0.000} C_DIS
LIN {X -190.159,Y +390.929,Z +0.000,A +0.000,E1 +46.494,E3 +186715.855,E4 +0.000} C_DIS
LIN {X -190.174,Y +383.973,Z +0.000,A +0.000,E1 +46.484,E3 +186724.748,E4 +0.000} C_DIS
LIN {X -190.200,Y +373.815,Z +0.000,A +0.000,E1 +46.448,E3 +186737.753,E4 +0.000} C_DIS
LIN {X -190.154,Y +361.003,Z +0.000,A +0.000,E1 +46.303,E3 +186754.247,E4 +0.000} C_DIS
LIN {X -189.772,Y +350.660,Z +0.000,A +0.049,E1 +45.996,E3 +186767.786,E4 +0.000} C_DIS
LIN {X -189.325,Y +346.917,Z +0.000,A +0.243,E1 +45.771,E3 +186772.855,E4 +0.000} C_DIS
LIN {X -188.196,Y +342.754,Z +0.000,A +1.966,E1 +45.249,E3 +186778.863,E4 +0.000} C_DIS
LIN {X -185.199,Y +337.023,Z +0.000,A +6.630,E1 +43.793,E3 +186788.237,E4 +0.000} C_DIS
LIN {X -181.141,Y +331.596,Z +0.000,A +12.274,E1 +41.569,E3 +186798.797,E4 +0.000} C_DIS
LIN {X -176.762,Y +326.804,Z +0.000,A +17.560,E1 +38.898,E3 +186810.221,E4 +0.000} C_DIS
LIN {X -172.184,Y +322.578,Z +0.000,A +19.859,E1 +36.197,E3 +186822.951,E4 +0.000} C_DIS
LIN {X -165.998,Y +317.874,Z +0.000,A +20.000,E1 +32.027,E3 +186842.709,E4 +0.000} C_DIS
LIN {X -160.137,Y +314.334,Z +0.000,A +20.000,E1 +26.368,E3 +186867.078,E4 +0.000} C_DIS
LIN {X -155.624,Y +312.245,Z +0.000,A +20.000,E1 +19.506,E3 +186895.754,E4 +0.000} C_DIS
LIN {X -153.557,Y +311.879,Z +0.000,A +20.000,E1 +11.113,E3 +186931.509,E4 +0.000} C_DIS
LIN {X -155.320,Y +313.348,Z +0.000,A +20.000,E1 +3.401,E3 +186964.693,E4 +0.000} C_DIS
LIN {X -160.005,Y +315.804,Z +0.000,A +20.000,E1 -4.720,E3 +186995.071,E4 +0.000} C_DIS
LIN {X -164.504,Y +318.255,Z +0.000,A +20.000,E1 -10.663,E3 +187014.440,E4 +0.000} C_DIS
LIN {X -170.340,Y +322.684,Z +0.000,A +20.000,E1 -17.457,E3 +187034.472,E4 +0.000} C_DIS
LIN {X -175.568,Y +329.106,Z +0.000,A +20.000,E1 -24.747,E3 +187051.706,E4 +0.000} C_DIS
LIN {X -184.074,Y +340.065,Z +0.000,A +20.000,E1 -33.664,E3 +187074.646,E4 +0.000} C_DIS
LIN {X -190.779,Y +351.388,Z +0.000,A +20.000,E1 -40.083,E3 +187092.424,E4 +0.000} C_DIS
LIN {X -195.254,Y +362.955,Z +0.000,A +20.000,E1 -44.515,E3 +187107.177,E4 +0.000} C_DIS
LIN {X -197.754,Y +374.780,Z +0.000,A +20.000,E1 -47.450,E3 +187120.599,E4 +0.000} C_DIS
LIN {X -198.310,Y +383.215,Z +0.000,A +19.956,E1 -48.698,E3 +187129.723,E4 +0.000} C_DIS
LIN {X -197.912,Y +391.275,Z +0.000,A +18.601,E1 -49.158,E3 +187138.441,E4 +0.000} C_DIS
LIN {X -196.679,Y +398.944,Z +0.000,A +13.989,E1 -48.784,E3 +187146.995,E4 +0.000} C_DIS
LIN {X -194.742,Y +406.288,Z +0.000,A +8.476,E1 -48.001,E3 +187155.678,E4 +0.000} C_DIS
LIN {X -192.748,Y +413.472,Z +0.000,A +3.905,E1 -47.267,E3 +187164.688,E4 +0.000} C_DIS
LIN {X -191.781,Y +419.162,Z +0.000,A +1.739,E1 -46.975,E3 +187171.956,E4 +0.000} C_DIS
LIN {X -190.795,Y +430.646,Z +0.000,A +0.152,E1 -46.707,E3 +187186.617,E4 +0.000} C_DIS
LIN {X -190.395,Y +441.145,Z +0.000,A +0.001,E1 -46.583,E3 +187200.010,E4 +0.000} C_DIS
LIN {X -190.239,Y +451.150,Z +0.000,A -0.000,E1 -46.528,E3 +187212.778,E4 +0.000} C_DIS
LIN {X -190.161,Y +465.026,Z +0.000,A -0.000,E1 -46.506,E3 +187230.493,E4 +0.000} C_DIS
LIN {X -190.142,Y +1057.148,Z +0.000,A -0.000,E1 -46.500,E3 +187986.699,E4 +0.000} C_DIS
LIN {X -190.147,Y +1068.924,Z +0.000,A -0.000,E1 -46.499,E3 +188001.740,E4 +0.000} C_DIS
LIN {X -190.159,Y +1079.072,Z +0.000,A -0.000,E1 -46.493,E3 +188014.705,E4 +0.000} C_DIS
LIN {X -190.174,Y +1086.028,Z +0.000,A -0.000,E1 -46.483,E3 +188023.599,E4 +0.000} C_DIS
LIN {X -190.200,Y +1096.186,Z +0.000,A -0.000,E1 -46.448,E3 +188036.603,E4 +0.000} C_DIS
LIN {X -190.154,Y +1108.998,Z +0.000,A -0.054,E1 -46.295,E3 +188053.098,E4 +0.000} C_DIS
LIN {X -189.772,Y +1119.341,Z +0.000,A -0.752,E1 -45.902,E3 +188066.636,E4 +0.000} C_DIS
LIN {X -189.097,Y +1124.276,Z +0.000,A -2.508,E1 -45.397,E3 +188073.368,E4 +0.000} C_DIS
LIN {X -187.410,Y +1129.069,Z +0.000,A -5.304,E1 -44.585,E3 +188080.541,E4 +0.000} C_DIS
LIN {X -183.899,Y +1134.873,Z +0.000,A -10.372,E1 -42.805,E3 +188090.547,E4 +0.000} C_DIS
LIN {X -179.711,Y +1140.065,Z +0.000,A -15.940,E1 -40.393,E3 +188101.333,E4 +0.000} C_DIS
LIN {X -176.763,Y +1143.197,Z +0.000,A -18.748,E1 -38.674,E3 +188109.071,E4 +0.000} C_DIS
LIN {X -172.185,Y +1147.423,Z +0.000,A -19.971,E1 -36.175,E3 +188121.801,E4 +0.000} C_DIS
LIN {X -165.999,Y +1152.127,Z +0.000,A -20.000,E1 -32.027,E3 +188141.559,E4 +0.000} C_DIS
LIN {X -160.138,Y +1155.667,Z +0.000,A -20.000,E1 -26.368,E3 +188165.929,E4 +0.000} C_DIS
LIN {X -155.625,Y +1157.756,Z +0.000,A -20.000,E1 -19.505,E3 +188194.605,E4 +0.000} C_DIS
LIN {X -153.552,Y +1158.113,Z +0.000,A -20.000,E1 -11.113,E3 +188230.356,E4 +0.000} C_DIS
LIN {X -156.311,Y +1155.540,Z +0.000,A -20.000,E1 -0.839,E3 +188273.716,E4 +0.000} C_DIS
LIN {X -161.281,Y +1151.851,Z +0.000,A -20.000,E1 +7.737,E3 +188303.615,E4 +0.000} C_DIS
LIN {X -167.493,Y +1147.157,Z +0.000,A -20.000,E1 +16.195,E3 +188328.054,E4 +0.000} C_DIS
LIN {X -173.235,Y +1142.221,Z +0.000,A -20.000,E1 +22.930,E3 +188345.356,E4 +0.000} C_DIS
LIN {X -181.123,Y +1133.734,Z +0.000,A -20.000,E1 +30.868,E3 +188366.112,E4 +0.000} C_DIS
LIN {X -189.654,Y +1120.856,Z +0.000,A -20.000,E1 +39.018,E3 +188388.126,E4 +0.000} C_DIS
LIN {X -195.246,Y +1107.046,Z +0.000,A -20.000,E1 +44.515,E3 +188406.028,E4 +0.000} C_DIS
LIN {X -198.051,Y +1092.368,Z +0.000,A -20.000,E1 +47.947,E3 +188422.554,E4 +0.000} C_DIS
LIN {X -198.143,Y +1081.370,Z +0.000,A -19.806,E1 +49.153,E3 +188434.415,E4 +0.000} C_DIS
LIN {X -197.177,Y +1073.569,Z +0.000,A -17.356,E1 +49.162,E3 +188442.999,E4 +0.000} C_DIS
LIN {X -195.448,Y +1066.139,Z +0.000,A -12.154,E1 +48.512,E3 +188451.594,E4 +0.000} C_DIS
LIN {X -193.346,Y +1058.941,Z +0.000,A -7.133,E1 +47.724,E3 +188460.474,E4 +0.000} C_DIS
LIN {X -191.781,Y +1050.839,Z +0.000,A -3.715,E1 +47.274,E3 +188470.807,E4 +0.000} C_DIS
LIN {X -190.795,Y +1039.355,Z +0.000,A -0.983,E1 +46.842,E3 +188485.467,E4 +0.000} C_DIS
LIN {X -190.395,Y +1028.856,Z +0.000,A -0.089,E1 +46.598,E3 +188498.861,E4 +0.000} C_DIS
LIN {X -190.239,Y +1018.851,Z +0.000,A -0.004,E1 +46.529,E3 +188511.629,E4 +0.000} C_DIS
LIN {X -190.161,Y +1004.975,Z +0.000,A +0.000,E1 +46.506,E3 +188529.343,E4 +0.000} C_DIS
LIN {X -190.142,Y +412.853,Z +0.000,A +0.000,E1 +46.501,E3 +189285.549,E4 +0.000} C_DIS
LIN {X -190.147,Y +401.077,Z +0.000,A +0.000,E1 +46.499,E3 +189300.590,E4 +0.000} C_DIS
LIN {X -190.159,Y +390.929,Z +0.000,A +0.000,E1 +46.494,E3 +189313.556,E4 +0.000} C_DIS
LIN {X -190.174,Y +383.973,Z +0.000,A +0.000,E1 +46.484,E3 +189322.449,E4 +0.000} C_DIS
LIN {X -190.200,Y +373.815,Z +0.000,A +0.000,E1 +46.448,E3 +189335.454,E4 +0.000} C_DIS
LIN {X -190.154,Y +361.003,Z +0.000,A +0.000,E1 +46.303,E3 +189351.948,E4 +0.000} C_DIS
LIN {X -189.772,Y +350.660,Z +0.000,A +0.049,E1 +45.996,E3 +189365.487,E4 +0.000} C_DIS
LIN {X -189.325,Y +346.917,Z +0.000,A +0.243,E1 +45.771,E3 +189370.556,E4 +0.000} C_DIS
LIN {X -188.196,Y +342.754,Z +0.000,A +1.966,E1 +45.249,E3 +189376.564,E4 +0.000} C_DIS
LIN {X -185.199,Y +337.023,Z +0.000,A +6.630,E1 +43.793,E3 +189385.938,E4 +0.000} C_DIS
LIN {X -181.141,Y +331.596,Z +0.000,A +12.274,E1 +41.569,E3 +189396.498,E4 +0.000} C_DIS
LIN {X -176.762,Y +326.804,Z +0.000,A +17.560,E1 +38.898,E3 +189407.922,E4 +0.000} C_DIS
LIN {X -172.184,Y +322.578,Z +0.000,A +19.859,E1 +36.197,E3 +189420.652,E4 +0.000} C_DIS
LIN {X -165.998,Y +317.874,Z +0.000,A +20.000,E1 +32.027,E3 +189440.410,E4 +0.000} C_DIS
LIN {X -160.137,Y +314.334,Z +0.000,A +20.000,E1 +26.368,E3 +189464.779,E4 +0.000} C_DIS
LIN {X -155.624,Y +312.245,Z +0.000,A +20.000,E1 +19.506,E3 +189493.455,E4 +0.000} C_DIS
LIN {X -153.557,Y +311.879,Z +0.000,A +20.000,E1 +11.113,E3 +189529.210,E4 +0.000} C_DIS
LIN {X -155.320,Y +313.348,Z +0.000,A +20.000,E1 +3.401,E3 +189562.394,E4 +0.000} C_DIS
LIN {X -160.005,Y +315.804,Z +0.000,A +20.000,E1 -4.720,E3 +189592.772,E4 +0.000} C_DIS
LIN {X -164.504,Y +318.255,Z +0.000,A +20.000,E1 -10.663,E3 +189612.141,E4 +0.000} C_DIS
LIN {X -170.340,Y +322.684,Z +0.000,A +20.000,E1 -17.457,E3 +189632.173,E4 +0.000} C_DIS
LIN {X -175.568,Y +329.106,Z +0.000,A +20.000,E1 -24.747,E3 +189649.407,E4 +0.000} C_DIS
LIN {X -184.074,Y +340.065,Z +0.000,A +20.000,E1 -33.664,E3 +189672.347,E4 +0.000} C_DIS
LIN {X -190.779,Y +351.388,Z +0.000,A +20.000,E1 -40.083,E3 +189690.125,E4 +0.000} C_DIS
LIN {X -195.254,Y +362.955,Z +0.000,A +20.000,E1 -44.515,E3 +189704.878,E4 +0.000} C_DIS
LIN {X -197.754,Y +374.780,Z +0.000,A +20.000,E1 -47.450,E3 +189718.300,E4 +0.000} C_DIS
LIN {X -198.310,Y +383.215,Z +0.000,A +19.956,E1 -48.698,E3 +189727.424,E4 +0.000} C_DIS
LIN {X -197.912,Y +391.275,Z +0.000,A +18.601,E1 -49.158,E3 +189736.142,E4 +0.000} C_DIS
LIN {X -196.679,Y +398.944,Z +0.000,A +13.989,E1 -48.784,E3 +189744.696,E4 +0.000} C_DIS
LIN {X -194.742,Y +406.288,Z +0.000,A +8.476,E1 -48.001,E3 +189753.379,E4 +0.000} C_DIS
LIN {X -192.748,Y +413.472,Z +0.000,A +3.905,E1 -47.267,E3 +189762.389,E4 +0.000} C_DIS
LIN {X -191.781,Y +419.162,Z +0.000,A +1.739,E1 -46.975,E3 +189769.657,E4 +0.000} C_DIS
LIN {X -190.795,Y +430.646,Z +0.000,A +0.152,E1 -46.707,E3 +189784.318,E4 +0.000} C_DIS
LIN {X -190.395,Y +441.145,Z +0.000,A +0.001,E1 -46.583,E3 +189797.711,E4 +0.000} C_DIS
LIN {X -190.239,Y +451.150,Z +0.000,A -0.000,E1 -46.528,E3 +189810.479,E4 +0.000} C_DIS
LIN {X -190.161,Y +465.026,Z +0.000,A -0.000,E1 -46.506,E3 +189828.194,E4 +0.000} C_DIS
LIN {X -190.142,Y +1057.148,Z +0.000,A -0.000,E1 -46.500,E3 +190584.400,E4 +0.000} C_DIS
LIN {X -190.147,Y +1068.924,Z +0.000,A -0.000,E1 -46.499,E3 +190599.441,E4 +0.000} C_DIS
LIN {X -190.159,Y +1079.072,Z +0.000,A -0.000,E1 -46.493,E3 +190612.406,E4 +0.000} C_DIS
LIN {X -190.174,Y +1086.028,Z +0.000,A -0.000,E1 -46.483,E3 +190621.300,E4 +0.000} C_DIS
LIN {X -190.200,Y +1096.186,Z +0.000,A -0.000,E1 -46.448,E3 +190634.304,E4 +0.000} C_DIS
LIN {X -190.154,Y +1108.998,Z +0.000,A -0.054,E1 -46.295,E3 +190650.799,E4 +0.000} C_DIS
LIN {X -189.772,Y +1119.341,Z +0.000,A -0.752,E1 -45.902,E3 +190664.337,E4 +0.000} C_DIS
LIN {X -189.097,Y +1124.276,Z +0.000,A -2.508,E1 -45.397,E3 +190671.069,E4 +0.000} C_DIS
LIN {X -187.410,Y +1129.069,Z +0.000,A -5.304,E1 -44.585,E3 +190678.242,E4 +0.000} C_DIS
LIN {X -183.899,Y +1134.873,Z +0.000,A -10.372,E1 -42.805,E3 +190688.248,E4 +0.000} C_DIS
LIN {X -179.711,Y +1140.065,Z +0.000,A -15.940,E1 -40.393,E3 +190699.034,E4 +0.000} C_DIS
LIN {X -176.763,Y +1143.197,Z +0.000,A -18.748,E1 -38.674,E3 +190706.772,E4 +0.000} C_DIS
LIN {X -172.185,Y +1147.423,Z +0.000,A -19.971,E1 -36.175,E3 +190719.502,E4 +0.000} C_DIS
LIN {X -165.999,Y +1152.127,Z +0.000,A -20.000,E1 -32.027,E3 +190739.260,E4 +0.000} C_DIS
LIN {X -160.138,Y +1155.667,Z +0.000,A -20.000,E1 -26.368,E3 +190763.630,E4 +0.000} C_DIS
LIN {X -155.625,Y +1157.756,Z +0.000,A -20.000,E1 -19.505,E3 +190792.306,E4 +0.000} C_DIS
LIN {X -153.552,Y +1158.113,Z +0.000,A -20.000,E1 -11.113,E3 +190828.057,E4 +0.000} C_DIS
LIN {X -156.311,Y +1155.540,Z +0.000,A -20.000,E1 -0.839,E3 +190871.417,E4 +0.000} C_DIS
LIN {X -161.281,Y +1151.851,Z +0.000,A -20.000,E1 +7.737,E3 +190901.316,E4 +0.000} C_DIS
LIN {X -167.493,Y +1147.157,Z +0.000,A -20.000,E1 +16.195,E3 +190925.755,E4 +0.000} C_DIS
LIN {X -173.235,Y +1142.221,Z +0.000,A -20.000,E1 +22.930,E3 +190943.057,E4 +0.000} C_DIS
LIN {X -181.123,Y +1133.734,Z +0.000,A -20.000,E1 +30.868,E3 +190963.813,E4 +0.000} C_DIS
LIN {X -189.654,Y +1120.856,Z +0.000,A -20.000,E1 +39.018,E3 +190985.827,E4 +0.000} C_DIS
LIN {X -195.246,Y +1107.046,Z +0.000,A -20.000,E1 +44.515,E3 +191003.729,E4 +0.000} C_DIS
LIN {X -198.051,Y +1092.368,Z +0.000,A -20.000,E1 +47.947,E3 +191020.255,E4 +0.000} C_DIS
LIN {X -198.143,Y +1081.370,Z +0.000,A -19.806,E1 +49.153,E3 +191032.116,E4 +0.000} C_DIS
LIN {X -197.177,Y +1073.569,Z +0.000,A -17.356,E1 +49.162,E3 +191040.700,E4 +0.000} C_DIS
LIN {X -195.448,Y +1066.139,Z +0.000,A -12.154,E1 +48.512,E3 +191049.295,E4 +0.000} C_DIS
LIN {X -193.346,Y +1058.941,Z +0.000,A -7.133,E1 +47.724,E3 +191058.175,E4 +0.000} C_DIS
LIN {X -191.781,Y +1050.839,Z +0.000,A -3.715,E1 +47.274,E3 +191068.508,E4 +0.000} C_DIS
LIN {X -190.795,Y +1039.355,Z +0.000,A -0.983,E1 +46.842,E3 +191083.168,E4 +0.000} C_DIS
LIN {X -190.395,Y +1028.856,Z +0.000,A -0.089,E1 +46.598,E3 +191096.562,E4 +0.000} C_DIS
LIN {X -190.239,Y +1018.851,Z +0.000,A -0.004,E1 +46.529,E3 +191109.330,E4 +0.000} C_DIS
LIN {X -190.161,Y +1004.975,Z +0.000,A +0.000,E1 +46.506,E3 +191127.044,E4 +0.000} C_DIS
LIN {X -190.142,Y +412.853,Z +0.000,A +0.000,E1 +46.501,E3 +191883.250,E4 +0.000} C_DIS
LIN {X -190.147,Y +401.077,Z +0.000,A +0.000,E1 +46.499,E3 +191898.291,E4 +0.000} C_DIS
LIN {X -190.159,Y +390.929,Z +0.000,A +0.000,E1 +46.494,E3 +191911.257,E4 +0.000} C_DIS
LIN {X -190.174,Y +383.973,Z +0.000,A +0.000,E1 +46.484,E3 +191920.150,E4 +0.000} C_DIS
LIN {X -190.200,Y +373.815,Z +0.000,A +0.000,E1 +46.448,E3 +191933.155,E4 +0.000} C_DIS
LIN {X -190.154,Y +361.003,Z +0.000,A +0.000,E1 +46.303,E3 +191949.649,E4 +0.000} C_DIS
LIN {X -189.772,Y +350.660,Z +0.000,A +0.049,E1 +45.996,E3 +191963.188,E4 +0.000} C_DIS
LIN {X -189.325,Y +346.917,Z +0.000,A +0.243,E1 +45.771,E3 +191968.257,E4 +0.000} C_DIS
LIN {X -188.196,Y +342.754,Z +0.000,A +1.966,E1 +45.249,E3 +191974.265,E4 +0.000} C_DIS
LIN {X -185.199,Y +337.023,Z +0.000,A +6.630,E1 +43.793,E3 +191983.639,E4 +0.000} C_DIS
LIN {X -181.141,Y +331.596,Z +0.000,A +12.274,E1 +41.569,E3 +191994.199,E4 +0.000} C_DIS
LIN {X -176.762,Y +326.804,Z +0.000,A +17.560,E1 +38.898,E3 +192005.623,E4 +0.000} C_DIS
LIN {X -172.184,Y +322.578,Z +0.000,A +19.859,E1 +36.197,E3 +192018.353,E4 +0.000} C_DIS
LIN {X -165.998,Y +317.874,Z +0.000,A +20.000,E1 +32.027,E3 +192038.111,E4 +0.000} C_DIS
LIN {X -160.137,Y +314.334,Z +0.000,A +20.000,E1 +26.368,E3 +192062.480,E4 +0.000} C_DIS
LIN {X -155.624,Y +312.245,Z +0.000,A +20.000,E1 +19.506,E3 +192091.156,E4 +0.000} C_DIS
LIN {X -153.557,Y +311.879,Z +0.000,A +20.000,E1 +11.113,E3 +192126.911,E4 +0.000} C_DIS
LIN {X -155.320,Y +313.348,Z +0.000,A +20.000,E1 +3.401,E3 +192160.095,E4 +0.000} C_DIS
LIN {X -160.005,Y +315.804,Z +0.000,A +20.000,E1 -4.720,E3 +192190.473,E4 +0.000} C_DIS
LIN {X -164.504,Y +318.255,Z +0.000,A +20.000,E1 -10.663,E3 +192209.842,E4 +0.000} C_DIS
LIN {X -170.340,Y +322.684,Z +0.000,A +20.000,E1 -17.457,E3 +192229.874,E4 +0.000} C_DIS
LIN {X -175.568,Y +329.106,Z +0.000,A +20.000,E1 -24.747,E3 +192247.108,E4 +0.000} C_DIS
LIN {X -184.074,Y +340.065,Z +0.000,A +20.000,E1 -33.664,E3 +192270.048,E4 +0.000} C_DIS
LIN {X -190.779,Y +351.388,Z +0.000,A +20.000,E1 -40.083,E3 +192287.826,E4 +0.000} C_DIS
LIN {X -195.254,Y +362.955,Z +0.000,A +20.000,E1 -44.515,E3 +192302.579,E4 +0.000} C_DIS
LIN {X -197.754,Y +374.780,Z +0.000,A +20.000,E1 -47.450,E3 +192316.001,E4 +0.000} C_DIS
LIN {X -198.310,Y +383.215,Z +0.000,A +19.956,E1 -48.698,E3 +192325.125,E4 +0.000} C_DIS
LIN {X -197.912,Y +391.275,Z +0.000,A +18.601,E1 -49.158,E3 +192333.843,E4 +0.000} C_DIS
LIN {X -196.679,Y +398.944,Z +0.000,A +13.989,E1 -48.784,E3 +192342.397,E4 +0.000} C_DIS
LIN {X -194.742,Y +406.288,Z +0.000,A +8.476,E1 -48.001,E3 +192351.080,E4 +0.000} C_DIS
LIN {X -192.748,Y +413.472,Z +0.000,A +3.905,E1 -47.267,E3 +192360.090,E4 +0.000} C_DIS
LIN {X -191.781,Y +419.162,Z +0.000,A +1.739,E1 -46.975,E3 +192367.358,E4 +0.000} C_DIS
LIN {X -190.795,Y +430.646,Z +0.000,A +0.152,E1 -46.707,E3 +192382.019,E4 +0.000} C_DIS
LIN {X -190.395,Y +441.145,Z +0.000,A +0.001,E1 -46.583,E3 +192395.412,E4 +0.000} C_DIS
LIN {X -190.239,Y +451.150,Z +0.000,A -0.000,E1 -46.528,E3 +192408.180,E4 +0.000} C_DIS
LIN {X -190.161,Y +465.026,Z +0.000,A -0.000,E1 -46.506,E3 +192425.895,E4 +0.000} C_DIS
LIN {X -190.142,Y +1057.148,Z +0.000,A -0.000,E1 -46.500,E3 +193182.101,E4 +0.000} C_DIS
LIN {X -190.147,Y +1068.924,Z +0.000,A -0.000,E1 -46.499,E3 +193197.142,E4 +0.000} C_DIS
LIN {X -190.159,Y +1079.072,Z +0.000,A -0.000,E1 -46.493,E3 +193210.107,E4 +0.000} C_DIS
LIN {X -190.174,Y +1086.028,Z +0.000,A -0.000,E1 -46.483,E3 +193219.001,E4 +0.000} C_DIS
LIN {X -190.200,Y +1096.186,Z +0.000,A -0.000,E1 -46.448,E3 +193232.005,E4 +0.000} C_DIS
LIN {X -190.154,Y +1108.998,Z +0.000,A -0.054,E1 -46.295,E3 +193248.500,E4 +0.000} C_DIS
LIN {X -189.772,Y +1119.341,Z +0.000,A -0.752,E1 -45.902,E3 +193262.038,E4 +0.000} C_DIS
LIN {X -189.097,Y +1124.276,Z +0.000,A -2.508,E1 -45.397,E3 +193268.770,E4 +0.000} C_DIS
LIN {X -187.410,Y +1129.069,Z +0.000,A -5.304,E1 -44.585,E3 +193275.943,E4 +0.000} C_DIS
LIN {X -183.899,Y +1134.873,Z +0.000,A -10.372,E1 -42.805,E3 +193285.949,E4 +0.000} C_DIS
LIN {X -179.711,Y +1140.065,Z +0.000,A -15.940,E1 -40.393,E3 +193296.735,E4 +0.000} C_DIS
LIN {X -176.763,Y +1143.197,Z +0.000,A -18.748,E1 -38.674,E3 +193304.473,E4 +0.000} C_DIS
LIN {X -172.185,Y +1147.423,Z +0.000,A -19.971,E1 -36.175,E3 +193317.203,E4 +0.000} C_DIS
LIN {X -165.999,Y +1152.127,Z +0.000,A -20.000,E1 -32.027,E3 +193336.961,E4 +0.000} C_DIS
LIN {X -160.138,Y +1155.667,Z +0.000,A -20.000,E1 -26.368,E3 +193361.331,E4 +0.000} C_DIS
LIN {X -155.625,Y +1157.756,Z +0.000,A -20.000,E1 -19.505,E3 +193390.007,E4 +0.000} C_DIS
LIN {X -153.552,Y +1158.113,Z +0.000,A -20.000,E1 -11.113,E3 +193425.758,E4 +0.000} C_DIS
LIN {X -156.311,Y +1155.540,Z +0.000,A -20.000,E1 -0.839,E3 +193469.118,E4 +0.000} C_DIS
LIN {X -161.281,Y +1151.851,Z +0.000,A -20.000,E1 +7.737,E3 +193499.017,E4 +0.000} C_DIS
LIN {X -167.493,Y +1147.157,Z +0.000,A -20.000,E1 +16.195,E3 +193523.456,E4 +0.000} C_DIS
LIN {X -173.235,Y +1142.221,Z +0.000,A -20.000,E1 +22.930,E3 +193540.758,E4 +0.000} C_DIS
LIN {X -181.123,Y +1133.734,Z +0.000,A -20.000,E1 +30.868,E3 +193561.514,E4 +0.000} C_DIS
LIN {X -189.654,Y +1120.856,Z +0.000,A -20.000,E1 +39.018,E3 +193583.528,E4 +0.000} C_DIS
LIN {X -195.246,Y +1107.046,Z +0.000,A -20.000,E1 +44.515,E3 +193601.430,E4 +0.000} C_DIS
LIN {X -198.051,Y +1092.368,Z +0.000,A -20.000,E1 +47.947,E3 +193617.956,E4 +0.000} C_DIS
LIN {X -198.143,Y +1081.370,Z +0.000,A -19.806,E1 +49.153,E3 +193629.817,E4 +0.000} C_DIS
LIN {X -197.177,Y +1073.569,Z +0.000,A -17.356,E1 +49.162,E3 +193638.401,E4 +0.000} C_DIS
LIN {X -195.448,Y +1066.139,Z +0.000,A -12.154,E1 +48.512,E3 +193646.996,E4 +0.000} C_DIS
LIN {X -193.346,Y +1058.941,Z +0.000,A -7.133,E1 +47.724,E3 +193655.876,E4 +0.000} C_DIS
LIN {X -191.781,Y +1050.839,Z +0.000,A -3.715,E1 +47.274,E3 +193666.209,E4 +0.000} C_DIS
LIN {X -190.795,Y +1039.355,Z +0.000,A -0.983,E1 +46.842,E3 +193680.869,E4 +0.000} C_DIS
LIN {X -190.395,Y +1028.856,Z +0.000,A -0.089,E1 +46.598,E3 +193694.263,E4 +0.000} C_DIS
LIN {X -190.239,Y +1018.851,Z +0.000,A -0.004,E1 +46.529,E3 +193707.031,E4 +0.000} C_DIS
LIN {X -190.161,Y +1004.975,Z +0.000,A +0.000,E1 +46.506,E3 +193724.745,E4 +0.000} C_DIS
LIN {X -190.142,Y +412.853,Z +0.000,A +0.000,E1 +46.501,E3 +194480.951,E4 +0.000} C_DIS
LIN {X -190.147,Y +401.077,Z +0.000,A +0.000,E1 +46.499,E3 +194495.992,E4 +0.000} C_DIS
LIN {X -190.159,Y +390.929,Z +0.000,A +0.000,E1 +46.494,E3 +194508.958,E4 +0.000} C_DIS
LIN {X -190.174,Y +383.973,Z +0.000,A +0.000,E1 +46.484,E3 +194517.851,E4 +0.000} C_DIS
LIN {X -190.200,Y +373.815,Z +0.000,A +0.000,E1 +46.448,E3 +194530.856,E4 +0.000} C_DIS
LIN {X -190.154,Y +361.003,Z +0.000,A +0.000,E1 +46.303,E3 +194547.350,E4 +0.000} C_DIS
LIN {X -189.772,Y +350.660,Z +0.000,A +0.049,E1 +45.996,E3 +194560.889,E4 +0.000} C_DIS
LIN {X -189.325,Y +346.917,Z +0.000,A +0.243,E1 +45.771,E3 +194565.958,E4 +0.000} C_DIS
LIN {X -188.196,Y +342.754,Z +0.000,A +1.966,E1 +45.249,E3 +194571.966,E4 +0.000} C_DIS
LIN {X -185.199,Y +337.023,Z +0.000,A +6.630,E1 +43.793,E3 +194581.340,E4 +0.000} C_DIS
LIN {X -181.141,Y +331.596,Z +0.000,A +12.274,E1 +41.569,E3 +194591.900,E4 +0.000} C_DIS
LIN {X -176.762,Y +326.804,Z +0.000,A +17.560,E1 +38.898,E3 +194603.324,E4 +0.000} C_DIS
LIN {X -172.184,Y +322.578,Z +0.000,A +19.859,E1 +36.197,E3 +194616.054,E4 +0.000} C_DIS
LIN {X -165.998,Y +317.874,Z +0.000,A +20.000,E1 +32.027,E3 +194635.812,E4 +0.000} C_DIS
LIN {X -160.137,Y +314.334,Z +0.000,A +20.000,E1 +26.368,E3 +194660.181,E4 +0.000} C_DIS
LIN {X -155.624,Y +312.245,Z +0.000,A +20.000,E1 +19.506,E3 +194688.857,E4 +0.000} C_DIS
LIN {X -153.557,Y +311.879,Z +0.000,A +20.000,E1 +11.113,E3 +194724.612,E4 +0.000} C_DIS
LIN {X -155.320,Y +313.348,Z +0.000,A +20.000,E1 +3.401,E3 +194757.796,E4 +0.000} C_DIS
LIN {X -160.005,Y +315.804,Z +0.000,A +20.000,E1 -4.720,E3 +194788.174,E4 +0.000} C_DIS
LIN {X -164.504,Y +318.255,Z +0.000,A +20.000,E1 -10.663,E3 +194807.543,E4 +0.000} C_DIS
LIN {X -170.340,Y +322.684,Z +0.000,A +20.000,E1 -17.457,E3 +194827.575,E4 +0.000} C_DIS
LIN {X -175.568,Y +329.106,Z +0.000,A +20.000,E1 -24.747,E3 +194844.809,E4 +0.000} C_DIS
LIN {X -184.074,Y +340.065,Z +0.000,A +20.000,E1 -33.664,E3 +194867.749,E4 +0.000} C_DIS
LIN {X -190.779,Y +351.388,Z +0.000,A +20.000,E1 -40.083,E3 +194885.527,E4 +0.000} C_DIS
LIN {X -195.254,Y +362.955,Z +0.000,A +20.000,E1 -44.515,E3 +194900.280,E4 +0.000} C_DIS
LIN {X -197.754,Y +374.780,Z +0.000,A +20.000,E1 -47.450,E3 +194913.702,E4 +0.000} C_DIS
LIN {X -198.310,Y +383.215,Z +0.000,A +19.956,E1 -48.698,E3 +194922.826,E4 +0.000} C_DIS
LIN {X -197.912,Y +391.275,Z +0.000,A +18.601,E1 -49.158,E3 +194931.544,E4 +0.000} C_DIS
LIN {X -196.679,Y +398.944,Z +0.000,A +13.989,E1 -48.784,E3 +194940.098,E4 +0.000} C_DIS
LIN {X -194.742,Y +406.288,Z +0.000,A +8.476,E1 -48.001,E3 +194948.781,E4 +0.000} C_DIS
LIN {X -192.748,Y +413.472,Z +0.000,A +3.905,E1 -47.267,E3 +194957.791,E4 +0.000} C_DIS
LIN {X -191.781,Y +419.162,Z +0.000,A +1.739,E1 -46.975,E3 +194965.059,E4 +0.000} C_DIS
LIN {X -190.795,Y +430.646,Z +0.000,A +0.152,E1 -46.707,E3 +194979.720,E4 +0.000} C_DIS
LIN {X -190.395,Y +441.145,Z +0.000,A +0.001,E1 -46.583,E3 +194993.113,E4 +0.000} C_DIS
LIN {X -190.239,Y +451.150,Z +0.000,A -0.000,E1 -46.528,E3 +195005.881,E4 +0.000} C_DIS
LIN {X -190.161,Y +465.026,Z +0.000,A -0.000,E1 -46.506,E3 +195023.596,E4 +0.000} C_DIS
LIN {X -190.142,Y +1057.148,Z +0.000,A -0.000,E1 -46.500,E3 +195779.802,E4 +0.000} C_DIS
LIN {X -190.147,Y +1068.924,Z +0.000,A -0.000,E1 -46.499,E3 +195794.843,E4 +0.000} C_DIS
LIN {X -190.159,Y +1079.072,Z +0.000,A -0.000,E1 -46.493,E3 +195807.808,E4 +0.000} C_DIS
LIN {X -190.174,Y +1086.028,Z +0.000,A -0.000,E1 -46.483,E3 +195816.702,E4 +0.000} C_DIS
LIN {X -190.200,Y +1096.186,Z +0.000,A -0.000,E1 -46.448,E3 +195829.706,E4 +0.000} C_DIS
LIN {X -190.154,Y +1108.998,Z +0.000,A -0.054,E1 -46.295,E3 +195846.201,E4 +0.000} C_DIS
LIN {X -189.772,Y +1119.341,Z +0.000,A -0.752,E1 -45.902,E3 +195859.739,E4 +0.000} C_DIS
LIN {X -189.097,Y +1124.276,Z +0.000,A -2.508,E1 -45.397,E3 +195866.471,E4 +0.000} C_DIS
LIN {X -187.410,Y +1129.069,Z +0.000,A -5.304,E1 -44.585,E3 +195873.644,E4 +0.000} C_DIS
LIN {X -183.899,Y +1134.873,Z +0.000,A -10.372,E1 -42.805,E3 +195883.650,E4 +0.000} C_DIS
LIN {X -179.711,Y +1140.065,Z +0.000,A -15.940,E1 -40.393,E3 +195894.436,E4 +0.000} C_DIS
LIN {X -176.763,Y +1143.197,Z +0.000,A -18.748,E1 -38.674,E3 +195902.174,E4 +0.000} C_DIS
LIN {X -172.185,Y +1147.423,Z +0.000,A -19.971,E1 -36.175,E3 +195914.904,E4 +0.000} C_DIS
LIN {X -165.999,Y +1152.127,Z +0.000,A -20.000,E1 -32.027,E3 +195934.662,E4 +0.000} C_DIS
LIN {X -160.138,Y +1155.667,Z +0.000,A -20.000,E1 -26.368,E3 +195959.032,E4 +0.000} C_DIS
LIN {X -155.625,Y +1157.756,Z +0.000,A -20.000,E1 -19.505,E3 +195987.708,E4 +0.000} C_DIS
LIN {X -153.552,Y +1158.113,Z +0.000,A -20.000,E1 -11.113,E3 +196023.459,E4 +0.000} C_DIS
LIN {X -156.311,Y +1155.540,Z +0.000,A -20.000,E1 -0.839,E3 +196066.819,E4 +0.000} C_DIS
LIN {X -161.281,Y +1151.851,Z +0.000,A -20.000,E1 +7.737,E3 +196096.718,E4 +0.000} C_DIS
LIN {X -167.493,Y +1147.157,Z +0.000,A -20.000,E1 +16.195,E3 +196121.157,E4 +0.000} C_DIS
LIN {X -173.235,Y +1142.221,Z +0.000,A -20.000,E1 +22.930,E3 +196138.459,E4 +0.000} C_DIS
LIN {X -181.123,Y +1133.734,Z +0.000,A -20.000,E1 +30.868,E3 +196159.215,E4 +0.000} C_DIS
LIN {X -189.654,Y +1120.856,Z +0.000,A -20.000,E1 +39.018,E3 +196181.229,E4 +0.000} C_DIS
LIN {X -195.246,Y +1107.046,Z +0.000,A -20.000,E1 +44.515,E3 +196199.131,E4 +0.000} C_DIS
LIN {X -198.051,Y +1092.368,Z +0.000,A -20.000,E1 +47.947,E3 +196215.657,E4 +0.000} C_DIS
LIN {X -198.143,Y +1081.370,Z +0.000,A -19.806,E1 +49.153,E3 +196227.518,E4 +0.000} C_DIS
LIN {X -197.177,Y +1073.569,Z +0.000,A -17.356,E1 +49.162,E3 +196236.102,E4 +0.000} C_DIS
LIN {X -195.448,Y +1066.139,Z +0.000,A -12.154,E1 +48.512,E3 +196244.697,E4 +0.000} C_DIS
LIN {X -193.346,Y +1058.941,Z +0.000,A -7.133,E1 +47.724,E3 +196253.577,E4 +0.000} C_DIS
LIN {X -191.781,Y +1050.839,Z +0.000,A -3.715,E1 +47.274,E3 +196263.910,E4 +0.000} C_DIS
LIN {X -190.795,Y +1039.355,Z +0.000,A -0.983,E1 +46.842,E3 +196278.570,E4 +0.000} C_DIS
LIN {X -190.395,Y +1028.856,Z +0.000,A -0.089,E1 +46.598,E3 +196291.964,E4 +0.000} C_DIS
LIN {X -190.239,Y +1018.851,Z +0.000,A -0.004,E1 +46.529,E3 +196304.732,E4 +0.000} C_DIS
LIN {X -190.161,Y +1004.975,Z +0.000,A +0.000,E1 +46.506,E3 +196322.446,E4 +0.000} C_DIS
LIN {X -190.142,Y +412.853,Z +0.000,A +0.000,E1 +46.501,E3 +197078.652,E4 +0.000} C_DIS
LIN {X -190.147,Y +401.077,Z +0.000,A +0.000,E1 +46.499,E3 +197093.693,E4 +0.000} C_DIS
LIN {X -190.159,Y +390.929,Z +0.000,A +0.000,E1 +46.494,E3 +197106.659,E4 +0.000} C_DIS
LIN {X -190.174,Y +383.973,Z +0.000,A +0.000,E1 +46.484,E3 +197115.552,E4 +0.000} C_DIS
LIN {X -190.200,Y +373.815,Z +0.000,A +0.000,E1 +46.448,E3 +197128.557,E4 +0.000} C_DIS
LIN {X -190.154,Y +361.003,Z +0.000,A +0.000,E1 +46.303,E3 +197145.051,E4 +0.000} C_DIS
LIN {X -189.772,Y +350.660,Z +0.000,A +0.049,E1 +45.996,E3 +197158.590,E4 +0.000} C_DIS
LIN {X -189.325,Y +346.917,Z +0.000,A +0.243,E1 +45.771,E3 +197163.659,E4 +0.000} C_DIS
LIN {X -188.196,Y +342.754,Z +0.000,A +1.966,E1 +45.249,E3 +197169.667,E4 +0.000} C_DIS
LIN {X -185.199,Y +337.023,Z +0.000,A +6.630,E1 +43.793,E3 +197179.041,E4 +0.000} C_DIS
LIN {X -181.141,Y +331.596,Z +0.000,A +12.274,E1 +41.569,E3 +197189.601,E4 +0.000} C_DIS
LIN {X -176.762,Y +326.804,Z +0.000,A +17.560,E1 +38.898,E3 +197201.025,E4 +0.000} C_DIS
LIN {X -172.184,Y +322.578,Z +0.000,A +19.859,E1 +36.197,E3 +197213.755,E4 +0.000} C_DIS
LIN {X -165.998,Y +317.874,Z +0.000,A +20.000,E1 +32.027,E3 +197233.513,E4 +0.000} C_DIS
LIN {X -160.137,Y +314.334,Z +0.000,A +20.000,E1 +26.368,E3 +197257.882,E4 +0.000} C_DIS
LIN {X -155.624,Y +312.245,Z +0.000,A +20.000,E1 +19.506,E3 +197286.558,E4 +0.000} C_DIS
LIN {X -153.557,Y +311.879,Z +0.000,A +20.000,E1 +11.113,E3 +197322.313,E4 +0.000} C_DIS
LIN {X -155.320,Y +313.348,Z +0.000,A +20.000,E1 +3.401,E3 +197355.497,E4 +0.000} C_DIS
LIN {X -160.005,Y +315.804,Z +0.000,A +20.000,E1 -4.720,E3 +197385.875,E4 +0.000} C_DIS
LIN {X -164.504,Y +318.255,Z +0.000,A +20.000,E1 -10.663,E3 +197405.244,E4 +0.000} C_DIS
LIN {X -170.340,Y +322.684,Z +0.000,A +20.000,E1 -17.457,E3 +197425.276,E4 +0.000} C_DIS
LIN {X -175.568,Y +329.106,Z +0.000,A +20.000,E1 -24.747,E3 +197442.510,E4 +0.000} C_DIS
LIN {X -184.074,Y +340.065,Z +0.000,A +20.000,E1 -33.664,E3 +197465.450,E4 +0.000} C_DIS
LIN {X -190.779,Y +351.388,Z +0.000,A +20.000,E1 -40.083,E3 +197483.228,E4 +0.000} C_DIS
LIN {X -195.254,Y +362.955,Z +0.000,A +20.000,E1 -44.515,E3 +197497.981,E4 +0.000} C_DIS
LIN {X -197.754,Y +374.780,Z +0.000,A +20.000,E1 -47.450,E3 +197511.403,E4 +0.000} C_DIS
LIN {X -198.310,Y +383.215,Z +0.000,A +19.956,E1 -48.698,E3 +197520.527,E4 +0.000} C_DIS
LIN {X -197.912,Y +391.275,Z +0.000,A +18.601,E1 -49.158,E3 +197529.245,E4 +0.000} C_DIS
LIN {X -196.679,Y +398.944,Z +0.000,A +13.989,E1 -48.784,E3 +197537.799,E4 +0.000} C_DIS
LIN {X -194.742,Y +406.288,Z +0.000,A +8.476,E1 -48.001,E3 +197546.482,E4 +0.000} C_DIS
LIN {X -192.748,Y +413.472,Z +0.000,A +3.905,E1 -47.267,E3 +197555.492,E4 +0.000} C_DIS
LIN {X -191.781,Y +419.162,Z +0.000,A +1.739,E1 -46.975,E3 +197562.760,E4 +0.000} C_DIS
LIN {X -190.795,Y +430.646,Z +0.000,A +0.152,E1 -46.707,E3 +197577.421,E4 +0.000} C_DIS
LIN {X -190.395,Y +441.145,Z +0.000,A +0.001,E1 -46.583,E3 +197590.814,E4 +0.000} C_DIS
LIN {X -190.239,Y +451.150,Z +0.000,A -0.000,E1 -46.528,E3 +197603.582,E4 +0.000} C_DIS
LIN {X -190.161,Y +465.026,Z +0.000,A -0.000,E1 -46.506,E3 +197621.297,E4 +0.000} C_DIS
LIN {X -190.142,Y +1057.148,Z +0.000,A -0.000,E1 -46.500,E3 +198377.503,E4 +0.000} C_DIS
LIN {X -190.147,Y +1068.924,Z +0.000,A -0.000,E1 -46.499,E3 +198392.544,E4 +0.000} C_DIS
LIN {X -190.159,Y +1079.072,Z +0.000,A -0.000,E1 -46.493,E3 +198405.509,E4 +0.000} C_DIS
LIN {X -190.174,Y +1086.028,Z +0.000,A -0.000,E1 -46.483,E3 +198414.403,E4 +0.000} C_DIS
LIN {X -190.200,Y +1096.186,Z +0.000,A -0.000,E1 -46.448,E3 +198427.407,E4 +0.000} C_DIS
LIN {X -190.154,Y +1108.998,Z +0.000,A -0.054,E1 -46.295,E3 +198443.902,E4 +0.000} C_DIS
LIN {X -189.772,Y +1119.341,Z +0.000,A -0.752,E1 -45.902,E3 +198457.440,E4 +0.000} C_DIS
LIN {X -189.097,Y +1124.276,Z +0.000,A -2.508,E1 -45.397,E3 +198464.172,E4 +0.000} C_DIS
LIN {X -187.410,Y +1129.069,Z +0.000,A -5.304,E1 -44.585,E3 +198471.345,E4 +0.000} C_DIS
LIN {X -183.899,Y +1134.873,Z +0.000,A -10.372,E1 -42.805,E3 +198481.351,E4 +0.000} C_DIS
LIN {X -179.711,Y +1140.065,Z +0.000,A -15.940,E1 -40.393,E3 +198492.137,E4 +0.000} C_DIS
LIN {X -176.763,Y +1143.197,Z +0.000,A -18.748,E1 -38.674,E3 +198499.875,E4 +0.000} C_DIS
LIN {X -172.185,Y +1147.423,Z +0.000,A -19.971,E1 -36.175,E3 +198512.605,E4 +0.000} C_DIS
LIN {X -165.999,Y +1152.127,Z +0.000,A -20.000,E1 -32.027,E3 +198532.363,E4 +0.000} C_DIS
LIN {X -160.138,Y +1155.667,Z +0.000,A -20.000,E1 -26.368,E3 +198556.733,E4 +0.000} C_DIS
LIN {X -155.625,Y +1157.756,Z +0.000,A -20.000,E1 -19.505,E3 +198585.409,E4 +0.000} C_DIS
LIN {X -153.552,Y +1158.113,Z +0.000,A -20.000,E1 -11.113,E3 +198621.160,E4 +0.000} C_DIS
LIN {X -156.311,Y +1155.540,Z +0.000,A -20.000,E1 -0.839,E3 +198664.520,E4 +0.000} C_DIS
LIN {X -161.281,Y +1151.851,Z +0.000,A -20.000,E1 +7.737,E3 +198694.419,E4 +0.000} C_DIS
LIN {X -167.493,Y +1147.157,Z +0.000,A -20.000,E1 +16.195,E3 +198718.858,E4 +0.000} C_DIS
LIN {X -173.235,Y +1142.221,Z +0.000,A -20.000,E1 +22.930,E3 +198736.160,E4 +0.000} C_DIS
LIN {X -181.123,Y +1133.734,Z +0.000,A -20.000,E1 +30.868,E3 +198756.916,E4 +0.000} C_DIS
LIN {X -189.654,Y +1120.856,Z +0.000,A -20.000,E1 +39.018,E3 +198778.930,E4 +0.000} C_DIS
LIN {X -195.246,Y +1107.046,Z +0.000,A -20.000,E1 +44.515,E3 +198796.832,E4 +0.000} C_DIS
LIN {X -198.051,Y +1092.368,Z +0.000,A -20.000,E1 +47.947,E3 +198813.358,E4 +0.000} C_DIS
LIN {X -198.143,Y +1081.370,Z +0.000,A -19.806,E1 +49.153,E3 +198825.219,E4 +0.000} C_DIS
LIN {X -197.177,Y +1073.569,Z +0.000,A -17.356,E1 +49.162,E3 +198833.803,E4 +0.000} C_DIS
LIN {X -195.448,Y +1066.139,Z +0.000,A -12.154,E1 +48.512,E3 +198842.398,E4 +0.000} C_DIS
LIN {X -193.346,Y +1058.941,Z +0.000,A -7.133,E1 +47.724,E3 +198851.278,E4 +0.000} C_DIS
LIN {X -191.781,Y +1050.839,Z +0.000,A -3.715,E1 +47.274,E3 +198861.611,E4 +0.000} C_DIS
LIN {X -190.795,Y +1039.355,Z +0.000,A -0.983,E1 +46.842,E3 +198876.271,E4 +0.000} C_DIS
LIN {X -190.395,Y +1028.856,Z +0.000,A -0.089,E1 +46.598,E3 +198889.665,E4 +0.000} C_DIS
LIN {X -190.239,Y +1018.851,Z +0.000,A -0.004,E1 +46.529,E3 +198902.433,E4 +0.000} C_DIS
LIN {X -190.161,Y +1004.975,Z +0.000,A +0.000,E1 +46.506,E3 +198920.147,E4 +0.000} C_DIS
LIN {X -190.142,Y +412.853,Z +0.000,A +0.000,E1 +46.501,E3 +199676.353,E4 +0.000} C_DIS
LIN {X -190.147,Y +401.077,Z +0.000,A +0.000,E1 +46.499,E3 +199691.394,E4 +0.000} C_DIS
LIN {X -190.159,Y +390.929,Z +0.000,A +0.000,E1 +46.494,E3 +199704.360,E4 +0.000} C_DIS
LIN {X -190.174,Y +383.973,Z +0.000,A +0.000,E1 +46.484,E3 +199713.253,E4 +0.000} C_DIS
LIN {X -190.200,Y +373.815,Z +0.000,A +0.000,E1 +46.448,E3 +199726.258,E4 +0.000} C_DIS
LIN {X -190.154,Y +361.003,Z +0.000,A +0.000,E1 +46.303,E3 +199742.752,E4 +0.000} C_DIS
LIN {X -189.772,Y +350.660,Z +0.000,A +0.049,E1 +45.996,E3 +199756.291,E4 +0.000} C_DIS
LIN {X -189.325,Y +346.917,Z +0.000,A +0.243,E1 +45.771,E3 +199761.360,E4 +0.000} C_DIS
LIN {X -188.196,Y +342.754,Z +0.000,A +1.966,E1 +45.249,E3 +199767.368,E4 +0.000} C_DIS
LIN {X -185.199,Y +337.023,Z +0.000,A +6.630,E1 +43.793,E3 +199776.742,E4 +0.000} C_DIS
LIN {X -181.141,Y +331.596,Z +0.000,A +12.274,E1 +41.569,E3 +199787.302,E4 +0.000} C_DIS
LIN {X -176.762,Y +326.804,Z +0.000,A +17.560,E1 +38.898,E3 +199798.726,E4 +0.000} C_DIS
LIN {X -172.184,Y +322.578,Z +0.000,A +19.859,E1 +36.197,E3 +199811.456,E4 +0.000} C_DIS
LIN {X -165.998,Y +317.874,Z +0.000,A +20.000,E1 +32.027,E3 +199831.214,E4 +0.000} C_DIS
LIN {X -160.137,Y +314.334,Z +0.000,A +20.000,E1 +26.368,E3 +199855.583,E4 +0.000} C_DIS
LIN {X -155.624,Y +312.245,Z +0.000,A +20.000,E1 +19.506,E3 +199884.259,E4 +0.000} C_DIS
LIN {X -153.557,Y +311.879,Z +0.000,A +20.000,E1 +11.113,E3 +199920.014,E4 +0.000} C_DIS
LIN {X -155.320,Y +313.348,Z +0.000,A +20.000,E1 +3.401,E3 +199953.198,E4 +0.000} C_DIS
LIN {X -160.005,Y +315.804,Z +0.000,A +20.000,E1 -4.720,E3 +199983.576,E4 +0.000} C_DIS
LIN {X -164.504,Y +318.255,Z +0.000,A +20.000,E1 -10.663,E3 +200002.945,E4 +0.000} C_DIS
LIN {X -170.340,Y +322.684,Z +0.000,A +20.000,E1 -17.457,E3 +200022.977,E4 +0.000} C_DIS
LIN {X -175.568,Y +329.106,Z +0.000,A +20.000,E1 -24.747,E3 +200040.211,E4 +0.000} C_DIS
LIN {X -184.074,Y +340.065,Z +0.000,A +20.000,E1 -33.664,E3 +200063.151,E4 +0.000} C_DIS
LIN {X -190.779,Y +351.388,Z +0.000,A +20.000,E1 -40.083,E3 +200080.929,E4 +0.000} C_DIS
LIN {X -195.254,Y +362.955,Z +0.000,A +20.000,E1 -44.515,E3 +200095.682,E4 +0.000} C_DIS
LIN {X -197.754,Y +374.780,Z +0.000,A +20.000,E1 -47.450,E3 +200109.104,E4 +0.000} C_DIS
LIN {X -198.310,Y +383.215,Z +0.000,A +19.956,E1 -48.698,E3 +200118.228,E4 +0.000} C_DIS
LIN {X -197.912,Y +391.275,Z +0.000,A +18.601,E1 -49.158,E3 +200126.946,E4 +0.000} C_DIS
LIN {X -196.679,Y +398.944,Z +0.000,A +13.989,E1 -48.784,E3 +200135.500,E4 +0.000} C_DIS
LIN {X -194.742,Y +406.288,Z +0.000,A +8.476,E1 -48.001,E3 +200144.183,E4 +0.000} C_DIS
LIN {X -192.748,Y +413.472,Z +0.000,A +3.905,E1 -47.267,E3 +200153.193,E4 +0.000} C_DIS
LIN {X -191.781,Y +419.162,Z +0.000,A +1.739,E1 -46.975,E3 +200160.461,E4 +0.000} C_DIS
LIN {X -190.795,Y +430.646,Z +0.000,A +0.152,E1 -46.707,E3 +200175.122,E4 +0.000} C_DIS
LIN {X -190.395,Y +441.145,Z +0.000,A +0.001,E1 -46.583,E3 +200188.515,E4 +0.000} C_DIS
LIN {X -190.239,Y +451.150,Z +0.000,A -0.000,E1 -46.528,E3 +200201.283,E4 +0.000} C_DIS
LIN {X -190.161,Y +465.026,Z +0.000,A -0.000,E1 -46.506,E3 +200218.998,E4 +0.000} C_DIS
LIN {X -190.142,Y +1057.148,Z +0.000,A -0.000,E1 -46.500,E3 +200975.204,E4 +0.000} C_DIS
LIN {X -190.147,Y +1068.924,Z +0.000,A -0.000,E1 -46.499,E3 +200990.245,E4 +0.000} C_DIS
LIN {X -190.159,Y +1079.072,Z +0.000,A -0.000,E1 -46.493,E3 +201003.210,E4 +0.000} C_DIS
LIN {X -190.174,Y +1086.028,Z +0.000,A -0.000,E1 -46.483,E3 +201012.104,E4 +0.000} C_DIS
LIN {X -190.200,Y +1096.186,Z +0.000,A -0.000,E1 -46.448,E3 +201025.108,E4 +0.000} C_DIS
LIN {X -190.154,Y +1108.998,Z +0.000,A -0.054,E1 -46.295,E3 +201041.603,E4 +0.000} C_DIS
LIN {X -189.772,Y +1119.341,Z +0.000,A -0.752,E1 -45.902,E3 +201055.141,E4 +0.000} C_DIS
LIN {X -189.097,Y +1124.276,Z +0.000,A -2.508,E1 -45.397,E3 +201061.873,E4 +0.000} C_DIS
LIN {X -187.410,Y +1129.069,Z +0.000,A -5.304,E1 -44.585,E3 +201069.046,E4 +0.000} C_DIS
LIN {X -183.899,Y +1134.873,Z +0.000,A -10.372,E1 -42.805,E3 +201079.052,E4 +0.000} C_DIS
LIN {X -179.711,Y +1140.065,Z +0.000,A -15.940,E1 -40.393,E3 +201089.838,E4 +0.000} C_DIS
LIN {X -176.763,Y +1143.197,Z +0.000,A -18.748,E1 -38.674,E3 +201097.576,E4 +0.000} C_DIS
LIN {X -172.185,Y +1147.423,Z +0.000,A -19.971,E1 -36.175,E3 +201110.306,E4 +0.000} C_DIS
LIN {X -165.999,Y +1152.127,Z +0.000,A -20.000,E1 -32.027,E3 +201130.064,E4 +0.000} C_DIS
LIN {X -160.138,Y +1155.667,Z +0.000,A -20.000,E1 -26.368,E3 +201154.434,E4 +0.000} C_DIS
LIN {X -155.625,Y +1157.756,Z +0.000,A -20.000,E1 -19.505,E3 +201183.110,E4 +0.000} C_DIS
LIN {X -153.552,Y +1158.113,Z +0.000,A -20.000,E1 -11.113,E3 +201218.861,E4 +0.000} C_DIS
LIN {X -156.311,Y +1155.540,Z +0.000,A -20.000,E1 -0.839,E3 +201262.221,E4 +0.000} C_DIS
LIN {X -161.281,Y +1151.851,Z +0.000,A -20.000,E1 +7.737,E3 +201292.120,E4 +0.000} C_DIS
LIN {X -167.493,Y +1147.157,Z +0.000,A -20.000,E1 +16.195,E3 +201316.559,E4 +0.000} C_DIS
LIN {X -173.235,Y +1142.221,Z +0.000,A -20.000,E1 +22.930,E3 +201333.861,E4 +0.000} C_DIS
LIN {X -181.123,Y +1133.734,Z +0.000,A -20.000,E1 +30.868,E3 +201354.617,E4 +0.000} C_DIS
LIN {X -189.654,Y +1120.856,Z +0.000,A -20.000,E1 +39.018,E3 +201376.631,E4 +0.000} C_DIS
LIN {X -195.246,Y +1107.046,Z +0.000,A -20.000,E1 +44.515,E3 +201394.533,E4 +0.000} C_DIS
LIN {X -198.051,Y +1092.368,Z +0.000,A -20.000,E1 +47.947,E3 +201411.059,E4 +0.000} C_DIS
LIN {X -198.143,Y +1081.370,Z +0.000,A -19.806,E1 +49.153,E3 +201422.920,E4 +0.000} C_DIS
LIN {X -197.177,Y +1073.569,Z +0.000,A -17.356,E1 +49.162,E3 +201431.504,E4 +0.000} C_DIS
LIN {X -195.448,Y +1066.139,Z +0.000,A -12.154,E1 +48.512,E3 +201440.099,E4 +0.000} C_DIS
LIN {X -193.346,Y +1058.941,Z +0.000,A -7.133,E1 +47.724,E3 +201448.979,E4 +0.000} C_DIS
LIN {X -191.781,Y +1050.839,Z +0.000,A -3.715,E1 +47.274,E3 +201459.312,E4 +0.000} C_DIS
LIN {X -190.795,Y +1039.355,Z +0.000,A -0.983,E1 +46.842,E3 +201473.972,E4 +0.000} C_DIS
LIN {X -190.395,Y +1028.856,Z +0.000,A -0.089,E1 +46.598,E3 +201487.366,E4 +0.000} C_DIS
LIN {X -190.239,Y +1018.851,Z +0.000,A -0.004,E1 +46.529,E3 +201500.134,E4 +0.000} C_DIS
LIN {X -190.161,Y +1004.975,Z +0.000,A +0.000,E1 +46.506,E3 +201517.848,E4 +0.000} C_DIS
LIN {X -190.142,Y +412.853,Z +0.000,A +0.000,E1 +46.501,E3 +202274.054,E4 +0.000} C_DIS
LIN {X -190.147,Y +401.077,Z +0.000,A +0.000,E1 +46.499,E3 +202289.095,E4 +0.000} C_DIS
LIN {X -190.159,Y +390.929,Z +0.000,A +0.000,E1 +46.494,E3 +202302.061,E4 +0.000} C_DIS
LIN {X -190.174,Y +383.973,Z +0.000,A +0.000,E1 +46.484,E3 +202310.954,E4 +0.000} C_DIS
LIN {X -190.200,Y +373.815,Z +0.000,A +0.000,E1 +46.448,E3 +202323.959,E4 +0.000} C_DIS
LIN {X -190.154,Y +361.003,Z +0.000,A +0.000,E1 +46.303,E3 +202340.453,E4 +0.000} C_DIS
LIN {X -189.772,Y +350.660,Z +0.000,A +0.049,E1 +45.996,E3 +202353.992,E4 +0.000} C_DIS
LIN {X -189.325,Y +346.917,Z +0.000,A +0.243,E1 +45.771,E3 +202359.061,E4 +0.000} C_DIS
LIN {X -188.196,Y +342.754,Z +0.000,A +1.966,E1 +45.249,E3 +202365.069,E4 +0.000} C_DIS
LIN {X -185.199,Y +337.023,Z +0.000,A +6.630,E1 +43.793,E3 +202374.443,E4 +0.000} C_DIS
LIN {X -181.141,Y +331.596,Z +0.000,A +12.274,E1 +41.569,E3 +202385.003,E4 +0.000} C_DIS
LIN {X -176.762,Y +326.804,Z +0.000,A +17.560,E1 +38.898,E3 +202396.427,E4 +0.000} C_DIS
LIN {X -172.184,Y +322.578,Z +0.000,A +19.859,E1 +36.197,E3 +202409.157,E4 +0.000} C_DIS
LIN {X -165.998,Y +317.874,Z +0.000,A +20.000,E1 +32.027,E3 +202428.915,E4 +0.000} C_DIS
LIN {X -160.137,Y +314.334,Z +0.000,A +20.000,E1 +26.368,E3 +202453.284,E4 +0.000} C_DIS
LIN {X -155.624,Y +312.245,Z +0.000,A +20.000,E1 +19.506,E3 +202481.960,E4 +0.000} C_DIS
LIN {X -153.557,Y +311.879,Z +0.000,A +20.000,E1 +11.113,E3 +202517.715,E4 +0.000} C_DIS
LIN {X -155.320,Y +313.348,Z +0.000,A +20.000,E1 +3.401,E3 +202550.899,E4 +0.000} C_DIS
LIN {X -160.005,Y +315.804,Z +0.000,A +20.000,E1 -4.720,E3 +202581.277,E4 +0.000} C_DIS
LIN {X -164.504,Y +318.255,Z +0.000,A +20.000,E1 -10.663,E3 +202600.646,E4 +0.000} C_DIS
LIN {X -170.340,Y +322.684,Z +0.000,A +20.000,E1 -17.457,E3 +202620.678,E4 +0.000} C_DIS
LIN {X -175.568,Y +329.106,Z +0.000,A +20.000,E1 -24.747,E3 +202637.912,E4 +0.000} C_DIS
LIN {X -184.074,Y +340.065,Z +0.000,A +20.000,E1 -33.664,E3 +202660.852,E4 +0.000} C_DIS
LIN {X -190.779,Y +351.388,Z +0.000,A +20.000,E1 -40.083,E3 +202678.630,E4 +0.000} C_DIS
LIN {X -195.254,Y +362.955,Z +0.000,A +20.000,E1 -44.515,E3 +202693.383,E4 +0.000} C_DIS
LIN {X -197.754,Y +374.780,Z +0.000,A +20.000,E1 -47.450,E3 +202706.805,E4 +0.000} C_DIS
LIN {X -198.310,Y +383.215,Z +0.000,A +19.956,E1 -48.698,E3 +202715.929,E4 +0.000} C_DIS
LIN {X -197.912,Y +391.275,Z +0.000,A +18.601,E1 -49.158,E3 +202724.647,E4 +0.000} C_DIS
LIN {X -196.679,Y +398.944,Z +0.000,A +13.989,E1 -48.784,E3 +202733.201,E4 +0.000} C_DIS
LIN {X -194.742,Y +406.288,Z +0.000,A +8.476,E1 -48.001,E3 +202741.884,E4 +0.000} C_DIS
LIN {X -192.748,Y +413.472,Z +0.000,A +3.905,E1 -47.267,E3 +202750.894,E4 +0.000} C_DIS
LIN {X -191.781,Y +419.162,Z +0.000,A +1.739,E1 -46.975,E3 +202758.162,E4 +0.000} C_DIS
LIN {X -190.795,Y +430.646,Z +0.000,A +0.152,E1 -46.707,E3 +202772.823,E4 +0.000} C_DIS
LIN {X -190.395,Y +441.145,Z +0.000,A +0.001,E1 -46.583,E3 +202786.216,E4 +0.000} C_DIS
LIN {X -190.239,Y +451.150,Z +0.000,A -0.000,E1 -46.528,E3 +202798.984,E4 +0.000} C_DIS
LIN {X -190.161,Y +465.026,Z +0.000,A -0.000,E1 -46.506,E3 +202816.699,E4 +0.000} C_DIS
LIN {X -190.142,Y +1057.148,Z +0.000,A -0.000,E1 -46.500,E3 +203572.905,E4 +0.000} C_DIS
LIN {X -190.147,Y +1068.924,Z +0.000,A -0.000,E1 -46.499,E3 +203587.946,E4 +0.000} C_DIS
LIN {X -190.159,Y +1079.072,Z +0.000,A -0.000,E1 -46.493,E3 +203600.911,E4 +0.000} C_DIS
LIN {X -190.174,Y +1086.028,Z +0.000,A -0.000,E1 -46.483,E3 +203609.805,E4 +0.000} C_DIS
LIN {X -190.200,Y +1096.186,Z +0.000,A -0.000,E1 -46.448,E3 +203622.809,E4 +0.000} C_DIS
LIN {X -190.154,Y +1108.998,Z +0.000,A -0.054,E1 -46.295,E3 +203639.304,E4 +0.000} C_DIS
LIN {X -189.772,Y +1119.341,Z +0.000,A -0.752,E1 -45.902,E3 +203652.842,E4 +0.000} C_DIS
LIN {X -189.097,Y +1124.276,Z +0.000,A -2.508,E1 -45.397,E3 +203659.574,E4 +0.000} C_DIS
LIN {X -187.410,Y +1129.069,Z +0.000,A -5.304,E1 -44.585,E3 +203666.747,E4 +0.000} C_DIS
LIN {X -183.899,Y +1134.873,Z +0.000,A -10.372,E1 -42.805,E3 +203676.753,E4 +0.000} C_DIS
LIN {X -179.711,Y +1140.065,Z +0.000,A -15.940,E1 -40.393,E3 +203687.539,E4 +0.000} C_DIS
LIN {X -176.763,Y +1143.197,Z +0.000,A -18.748,E1 -38.674,E3 +203695.277,E4 +0.000} C_DIS
LIN {X -172.185,Y +1147.423,Z +0.000,A -19.971,E1 -36.175,E3 +203708.007,E4 +0.000} C_DIS
LIN {X -165.999,Y +1152.127,Z +0.000,A -20.000,E1 -32.027,E3 +203727.765,E4 +0.000} C_DIS
LIN {X -160.138,Y +1155.667,Z +0.000,A -20.000,E1 -26.368,E3 +203752.135,E4 +0.000} C_DIS
LIN {X -155.625,Y +1157.756,Z +0.000,A -20.000,E1 -19.505,E3 +203780.811,E4 +0.000} C_DIS
LIN {X -153.552,Y +1158.113,Z +0.000,A -20.000,E1 -11.113,E3 +203816.562,E4 +0.000} C_DIS
LIN {X -156.311,Y +1155.540,Z +0.000,A -20.000,E1 -0.839,E3 +203859.922,E4 +0.000} C_DIS
LIN {X -161.281,Y +1151.851,Z +0.000,A -20.000,E1 +7.737,E3 +203889.821,E4 +0.000} C_DIS
LIN {X -167.493,Y +1147.157,Z +0.000,A -20.000,E1 +16.195,E3 +203914.260,E4 +0.000} C_DIS
LIN {X -173.235,Y +1142.221,Z +0.000,A -20.000,E1 +22.930,E3 +203931.562,E4 +0.000} C_DIS
LIN {X -181.123,Y +1133.734,Z +0.000,A -20.000,E1 +30.868,E3 +203952.318,E4 +0.000} C_DIS
LIN {X -189.654,Y +1120.856,Z +0.000,A -20.000,E1 +39.018,E3 +203974.332,E4 +0.000} C_DIS
LIN {X -195.246,Y +1107.046,Z +0.000,A -20.000,E1 +44.515,E3 +203992.234,E4 +0.000} C_DIS
LIN {X -198.051,Y +1092.368,Z +0.000,A -20.000,E1 +47.947,E3 +204008.760,E4 +0.000} C_DIS
LIN {X -198.143,Y +1081.370,Z +0.000,A -19.806,E1 +49.153,E3 +204020.621,E4 +0.000} C_DIS
LIN {X -197.177,Y +1073.569,Z +0.000,A -17.356,E1 +49.162,E3 +204029.205,E4 +0.000} C_DIS
LIN {X -195.448,Y +1066.139,Z +0.000,A -12.154,E1 +48.512,E3 +204037.800,E4 +0.000} C_DIS
LIN {X -193.346,Y +1058.941,Z +0.000,A -7.133,E1 +47.724,E3 +204046.680,E4 +0.000} C_DIS
LIN {X -191.781,Y +1050.839,Z +0.000,A -3.715,E1 +47.274,E3 +204057.013,E4 +0.000} C_DIS
LIN {X -190.795,Y +1039.355,Z +0.000,A -0.983,E1 +46.842,E3 +204071.673,E4 +0.000} C_DIS
LIN {X -190.395,Y +1028.856,Z +0.000,A -0.089,E1 +46.598,E3 +204085.067,E4 +0.000} C_DIS
LIN {X -190.239,Y +1018.851,Z +0.000,A -0.004,E1 +46.529,E3 +204097.835,E4 +0.000} C_DIS
LIN {X -190.161,Y +1004.975,Z +0.000,A +0.000,E1 +46.506,E3 +204115.549,E4 +0.000} C_DIS
LIN {X -190.142,Y +412.853,Z +0.000,A +0.000,E1 +46.501,E3 +204871.755,E4 +0.000} C_DIS
LIN {X -190.147,Y +401.077,Z +0.000,A +0.000,E1 +46.499,E3 +204886.796,E4 +0.000} C_DIS
LIN {X -190.159,Y +390.929,Z +0.000,A +0.000,E1 +46.494,E3 +204899.762,E4 +0.000} C_DIS
LIN {X -190.174,Y +383.973,Z +0.000,A +0.000,E1 +46.484,E3 +204908.655,E4 +0.000} C_DIS
LIN {X -190.200,Y +373.815,Z +0.000,A +0.000,E1 +46.448,E3 +204921.660,E4 +0.000} C_DIS
LIN {X -190.154,Y +361.003,Z +0.000,A +0.000,E1 +46.303,E3 +204938.154,E4 +0.000} C_DIS
LIN {X -189.772,Y +350.660,Z +0.000,A +0.049,E1 +45.996,E3 +204951.693,E4 +0.000} C_DIS
LIN {X -189.325,Y +346.917,Z +0.000,A +0.243,E1 +45.771,E3 +204956.762,E4 +0.000} C_DIS
LIN {X -188.196,Y +342.754,Z +0.000,A +1.966,E1 +45.249,E3 +204962.770,E4 +0.000} C_DIS
LIN {X -185.199,Y +337.023,Z +0.000,A +6.630,E1 +43.793,E3 +204972.144,E4 +0.000} C_DIS
LIN {X -181.141,Y +331.596,Z +0.000,A +12.274,E1 +41.569,E3 +204982.704,E4 +0.000} C_DIS
LIN {X -176.762,Y +326.804,Z +0.000,A +17.560,E1 +38.898,E3 +204994.128,E4 +0.000} C_DIS
LIN {X -172.184,Y +322.578,Z +0.000,A +19.859,E1 +36.197,E3 +205006.858,E4 +0.000} C_DIS
LIN {X -165.998,Y +317.874,Z +0.000,A +20.000,E1 +32.027,E3 +205026.616,E4 +0.000} C_DIS
LIN {X -160.137,Y +314.334,Z +0.000,A +20.000,E1 +26.368,E3 +205050.985,E4 +0.000} C_DIS
LIN {X -155.624,Y +312.245,Z +0.000,A +20.000,E1 +19.506,E3 +205079.661,E4 +0.000} C_DIS
LIN {X -153.557,Y +311.879,Z +0.000,A +20.000,E1 +11.113,E3 +205115.416,E4 +0.000} C_DIS
LIN {X -155.320,Y +313.348,Z +0.000,A +20.000,E1 +3.401,E3 +205148.600,E4 +0.000} C_DIS
LIN {X -160.005,Y +315.804,Z +0.000,A +20.000,E1 -4.720,E3 +205178.978,E4 +0.000} C_DIS
LIN {X -164.504,Y +318.255,Z +0.000,A +20.000,E1 -10.663,E3 +205198.347,E4 +0.000} C_DIS
LIN {X -170.340,Y +322.684,Z +0.000,A +20.000,E1 -17.457,E3 +205218.379,E4 +0.000} C_DIS
LIN {X -175.568,Y +329.106,Z +0.000,A +20.000,E1 -24.747,E3 +205235.613,E4 +0.000} C_DIS
LIN {X -184.074,Y +340.065,Z +0.000,A +20.000,E1 -33.664,E3 +205258.553,E4 +0.000} C_DIS
LIN {X -190.779,Y +351.388,Z +0.000,A +20.000,E1 -40.083,E3 +205276.331,E4 +0.000} C_DIS
LIN {X -195.254,Y +362.955,Z +0.000,A +20.000,E1 -44.515,E3 +205291.084,E4 +0.000} C_DIS
LIN {X -197.754,Y +374.780,Z +0.000,A +20.000,E1 -47.450,E3 +205304.506,E4 +0.000} C_DIS
LIN {X -198.310,Y +383.215,Z +0.000,A +19.956,E1 -48.698,E3 +205313.630,E4 +0.000} C_DIS
LIN {X -197.912,Y +391.275,Z +0.000,A +18.601,E1 -49.158,E3 +205322.348,E4 +0.000} C_DIS
LIN {X -196.679,Y +398.944,Z +0.000,A +13.989,E1 -48.784,E3 +205330.902,E4 +0.000} C_DIS
LIN {X -194.742,Y +406.288,Z +0.000,A +8.476,E1 -48.001,E3 +205339.585,E4 +0.000} C_DIS
LIN {X -192.748,Y +413.472,Z +0.000,A +3.905,E1 -47.267,E3 +205348.595,E4 +0.000} C_DIS
LIN {X -191.781,Y +419.162,Z +0.000,A +1.739,E1 -46.975,E3 +205355.863,E4 +0.000} C_DIS
LIN {X -190.795,Y +430.646,Z +0.000,A +0.152,E1 -46.707,E3 +205370.524,E4 +0.000} C_DIS
LIN {X -190.395,Y +441.145,Z +0.000,A +0.001,E1 -46.583,E3 +205383.917,E4 +0.000} C_DIS
LIN {X -190.239,Y +451.150,Z +0.000,A -0.000,E1 -46.528,E3 +205396.685,E4 +0.000} C_DIS
LIN {X -190.161,Y +465.026,Z +0.000,A -0.000,E1 -46.506,E3 +205414.400,E4 +0.000} C_DIS
LIN {X -190.142,Y +1057.148,Z +0.000,A -0.000,E1 -46.500,E3 +206170.606,E4 +0.000} C_DIS
LIN {X -190.147,Y +1068.924,Z +0.000,A -0.000,E1 -46.499,E3 +206185.647,E4 +0.000} C_DIS
LIN {X -190.159,Y +1079.072,Z +0.000,A -0.000,E1 -46.493,E3 +206198.612,E4 +0.000} C_DIS
LIN {X -190.174,Y +1086.028,Z +0.000,A -0.000,E1 -46.483,E3 +206207.506,E4 +0.000} C_DIS
LIN {X -190.200,Y +1096.186,Z +0.000,A -0.000,E1 -46.448,E3 +206220.510,E4 +0.000} C_DIS
LIN {X -190.154,Y +1108.998,Z +0.000,A -0.054,E1 -46.295,E3 +206237.005,E4 +0.000} C_DIS
LIN {X -189.772,Y +1119.341,Z +0.000,A -0.752,E1 -45.902,E3 +206250.543,E4 +0.000} C_DIS
LIN {X -189.097,Y +1124.276,Z +0.000,A -2.508,E1 -45.397,E3 +206257.275,E4 +0.000} C_DIS
LIN {X -187.410,Y +1129.069,Z +0.000,A -5.304,E1 -44.585,E3 +206264.448,E4 +0.000} C_DIS
LIN {X -183.899,Y +1134.873,Z +0.000,A -10.372,E1 -42.805,E3 +206274.454,E4 +0.000} C_DIS
LIN {X -179.711,Y +1140.065,Z +0.000,A -15.940,E1 -40.393,E3 +206285.240,E4 +0.000} C_DIS
LIN {X -176.763,Y +1143.197,Z +0.000,A -18.748,E1 -38.674,E3 +206292.978,E4 +0.000} C_DIS
LIN {X -172.185,Y +1147.423,Z +0.000,A -19.971,E1 -36.175,E3 +206305.708,E4 +0.000} C_DIS
LIN {X -165.999,Y +1152.127,Z +0.000,A -20.000,E1 -32.027,E3 +206325.466,E4 +0.000} C_DIS
LIN {X -160.138,Y +1155.667,Z +0.000,A -20.000,E1 -26.368,E3 +206349.836,E4 +0.000} C_DIS
LIN {X -155.625,Y +1157.756,Z +0.000,A -20.000,E1 -19.505,E3 +206378.512,E4 +0.000} C_DIS
LIN {X -153.552,Y +1158.113,Z +0.000,A -20.000,E1 -11.113,E3 +206414.263,E4 +0.000} C_DIS
LIN {X -156.311,Y +1155.540,Z +0.000,A -20.000,E1 -0.839,E3 +206457.623,E4 +0.000} C_DIS
LIN {X -161.281,Y +1151.851,Z +0.000,A -20.000,E1 +7.737,E3 +206487.522,E4 +0.000} C_DIS
LIN {X -167.493,Y +1147.157,Z +0.000,A -20.000,E1 +16.195,E3 +206511.961,E4 +0.000} C_DIS
LIN {X -173.235,Y +1142.221,Z +0.000,A -20.000,E1 +22.930,E3 +206529.263,E4 +0.000} C_DIS
LIN {X -181.123,Y +1133.734,Z +0.000,A -20.000,E1 +30.868,E3 +206550.019,E4 +0.000} C_DIS
LIN {X -189.654,Y +1120.856,Z +0.000,A -20.000,E1 +39.018,E3 +206572.033,E4 +0.000} C_DIS
LIN {X -195.246,Y +1107.046,Z +0.000,A -20.000,E1 +44.515,E3 +206589.935,E4 +0.000} C_DIS
LIN {X -198.051,Y +1092.368,Z +0.000,A -20.000,E1 +47.947,E3 +206606.461,E4 +0.000} C_DIS
LIN {X -198.143,Y +1081.370,Z +0.000,A -19.806,E1 +49.153,E3 +206618.322,E4 +0.000} C_DIS
LIN {X -197.177,Y +1073.569,Z +0.000,A -17.356,E1 +49.162,E3 +206626.906,E4 +0.000} C_DIS
LIN {X -195.448,Y +1066.139,Z +0.000,A -12.154,E1 +48.512,E3 +206635.501,E4 +0.000} C_DIS
LIN {X -193.346,Y +1058.941,Z +0.000,A -7.133,E1 +47.724,E3 +206644.381,E4 +0.000} C_DIS
LIN {X -191.781,Y +1050.839,Z +0.000,A -3.715,E1 +47.274,E3 +206654.714,E4 +0.000} C_DIS
LIN {X -190.795,Y +1039.355,Z +0.000,A -0.983,E1 +46.842,E3 +206669.374,E4 +0.000} C_DIS
LIN {X -190.395,Y +1028.856,Z +0.000,A -0.089,E1 +46.598,E3 +206682.768,E4 +0.000} C_DIS
LIN {X -190.239,Y +1018.851,Z +0.000,A -0.004,E1 +46.529,E3 +206695.536,E4 +0.000} C_DIS
LIN {X -190.161,Y +1004.975,Z +0.000,A +0.000,E1 +46.506,E3 +206713.250,E4 +0.000} C_DIS
LIN {X -190.142,Y +412.853,Z +0.000,A +0.000,E1 +46.501,E3 +207469.456,E4 +0.000} C_DIS
LIN {X -190.147,Y +401.077,Z +0.000,A +0.000,E1 +46.499,E3 +207484.497,E4 +0.000} C_DIS
LIN {X -190.159,Y +390.929,Z +0.000,A +0.000,E1 +46.494,E3 +207497.463,E4 +0.000} C_DIS
LIN {X -190.174,Y +383.973,Z +0.000,A +0.000,E1 +46.484,E3 +207506.356,E4 +0.000} C_DIS
LIN {X -190.200,Y +373.815,Z +0.000,A +0.000,E1 +46.448,E3 +207519.361,E4 +0.000} C_DIS
LIN {X -190.154,Y +361.003,Z +0.000,A +0.000,E1 +46.303,E3 +207535.855,E4 +0.000} C_DIS
LIN {X -189.772,Y +350.660,Z +0.000,A +0.049,E1 +45.996,E3 +207549.394,E4 +0.000} C_DIS
LIN {X -189.325,Y +346.917,Z +0.000,A +0.243,E1 +45.771,E3 +207554.463,E4 +0.000} C_DIS
LIN {X -188.196,Y +342.754,Z +0.000,A +1.966,E1 +45.249,E3 +207560.471,E4 +0.000} C_DIS
LIN {X -185.199,Y +337.023,Z +0.000,A +6.630,E1 +43.793,E3 +207569.845,E4 +0.000} C_DIS
LIN {X -181.141,Y +331.596,Z +0.000,A +12.274,E1 +41.569,E3 +207580.405,E4 +0.000} C_DIS
LIN {X -176.762,Y +326.804,Z +0.000,A +17.560,E1 +38.898,E3 +207591.829,E4 +0.000} C_DIS
LIN {X -172.184,Y +322.578,Z +0.000,A +19.859,E1 +36.197,E3 +207604.559,E4 +0.000} C_DIS
LIN {X -165.998,Y +317.874,Z +0.000,A +20.000,E1 +32.027,E3 +207624.317,E4 +0.000} C_DIS
LIN {X -160.137,Y +314.334,Z +0.000,A +20.000,E1 +26.368,E3 +207648.686,E4 +0.000} C_DIS
LIN {X -155.624,Y +312.245,Z +0.000,A +20.000,E1 +19.506,E3 +207677.362,E4 +0.000} C_DIS
LIN {X -153.557,Y +311.879,Z +0.000,A +20.000,E1 +11.113,E3 +207713.117,E4 +0.000} C_DIS
LIN {X -155.320,Y +313.348,Z +0.000,A +20.000,E1 +3.401,E3 +207746.301,E4 +0.000} C_DIS
LIN {X -160.005,Y +315.804,Z +0.000,A +20.000,E1 -4.720,E3 +207776.679,E4 +0.000} C_DIS
LIN {X -164.504,Y +318.255,Z +0.000,A +20.000,E1 -10.663,E3 +207796.048,E4 +0.000} C_DIS
LIN {X -170.340,Y +322.684,Z +0.000,A +20.000,E1 -17.457,E3 +207816.080,E4 +0.000} C_DIS
LIN {X -175.568,Y +329.106,Z +0.000,A +20.000,E1 -24.747,E3 +207833.314,E4 +0.000} C_DIS
LIN {X -184.074,Y +340.065,Z +0.000,A +20.000,E1 -33.664,E3 +207856.254,E4 +0.000} C_DIS
LIN {X -190.779,Y +351.388,Z +0.000,A +20.000,E1 -40.083,E3 +207874.032,E4 +0.000} C_DIS
LIN {X -195.254,Y +362.955,Z +0.000,A +20.000,E1 -44.515,E3 +207888.785,E4 +0.000} C_DIS
LIN {X -197.754,Y +374.780,Z +0.000,A +20.000,E1 -47.450,E3 +207902.207,E4 +0.000} C_DIS
LIN {X -198.310,Y +383.215,Z +0.000,A +19.956,E1 -48.698,E3 +207911.331,E4 +0.000} C_DIS
LIN {X -197.912,Y +391.275,Z +0.000,A +18.601,E1 -49.158,E3 +207920.049,E4 +0.000} C_DIS
LIN {X -196.679,Y +398.944,Z +0.000,A +13.989,E1 -48.784,E3 +207928.603,E4 +0.000} C_DIS
LIN {X -194.742,Y +406.288,Z +0.000,A +8.476,E1 -48.001,E3 +207937.286,E4 +0.000} C_DIS
LIN {X -192.748,Y +413.472,Z +0.000,A +3.905,E1 -47.267,E3 +207946.296,E4 +0.000} C_DIS
LIN {X -191.781,Y +419.162,Z +0.000,A +1.739,E1 -46.975,E3 +207953.564,E4 +0.000} C_DIS
LIN {X -190.795,Y +430.646,Z +0.000,A +0.152,E1 -46.707,E3 +207968.225,E4 +0.000} C_DIS
LIN {X -190.395,Y +441.145,Z +0.000,A +0.001,E1 -46.583,E3 +207981.618,E4 +0.000} C_DIS
LIN {X -190.239,Y +451.150,Z +0.000,A -0.000,E1 -46.528,E3 +207994.386,E4 +0.000} C_DIS
LIN {X -190.161,Y +465.026,Z +0.000,A -0.000,E1 -46.506,E3 +208012.101,E4 +0.000} C_DIS
LIN {X -190.142,Y +1057.148,Z +0.000,A -0.000,E1 -46.500,E3 +208768.307,E4 +0.000} C_DIS
LIN {X -190.147,Y +1068.924,Z +0.000,A -0.000,E1 -46.499,E3 +208783.348,E4 +0.000} C_DIS
LIN {X -190.159,Y +1079.072,Z +0.000,A -0.000,E1 -46.493,E3 +208796.313,E4 +0.000} C_DIS
LIN {X -190.174,Y +1086.028,Z +0.000,A -0.000,E1 -46.483,E3 +208805.207,E4 +0.000} C_DIS
LIN {X -190.200,Y +1096.186,Z +0.000,A -0.000,E1 -46.448,E3 +208818.211,E4 +0.000} C_DIS
LIN {X -190.154,Y +1108.998,Z +0.000,A -0.054,E1 -46.295,E3 +208834.706,E4 +0.000} C_DIS
LIN {X -189.772,Y +1119.341,Z +0.000,A -0.752,E1 -45.902,E3 +208848.244,E4 +0.000} C_DIS
LIN {X -189.097,Y +1124.276,Z +0.000,A -2.508,E1 -45.397,E3 +208854.976,E4 +0.000} C_DIS
LIN {X -187.410,Y +1129.069,Z +0.000,A -5.304,E1 -44.585,E3 +208862.149,E4 +0.000} C_DIS
LIN {X -183.899,Y +1134.873,Z +0.000,A -10.372,E1 -42.805,E3 +208872.155,E4 +0.000} C_DIS
LIN {X -179.711,Y +1140.065,Z +0.000,A -15.940,E1 -40.393,E3 +208882.941,E4 +0.000} C_DIS
LIN {X -176.763,Y +1143.197,Z +0.000,A -18.748,E1 -38.674,E3 +208890.679,E4 +0.000} C_DIS
LIN {X -172.185,Y +1147.423,Z +0.000,A -19.971,E1 -36.175,E3 +208903.409,E4 +0.000} C_DIS
LIN {X -165.999,Y +1152.127,Z +0.000,A -20.000,E1 -32.027,E3 +208923.167,E4 +0.000} C_DIS
LIN {X -160.138,Y +1155.667,Z +0.000,A -20.000,E1 -26.368,E3 +208947.537,E4 +0.000} C_DIS
LIN {X -155.625,Y +1157.756,Z +0.000,A -20.000,E1 -19.505,E3 +208976.213,E4 +0.000} C_DIS
LIN {X -153.552,Y +1158.113,Z +0.000,A -20.000,E1 -11.113,E3 +209011.964,E4 +0.000} C_DIS
LIN {X -156.311,Y +1155.540,Z +0.000,A -20.000,E1 -0.839,E3 +209055.324,E4 +0.000} C_DIS
LIN {X -161.281,Y +1151.851,Z +0.000,A -20.000,E1 +7.737,E3 +209085.223,E4 +0.000} C_DIS
LIN {X -167.493,Y +1147.157,Z +0.000,A -20.000,E1 +16.195,E3 +209109.662,E4 +0.000} C_DIS
LIN {X -173.235,Y +1142.221,Z +0.000,A -20.000,E1 +22.930,E3 +209126.964,E4 +0.000} C_DIS
LIN {X -181.123,Y +1133.734,Z +0.000,A -20.000,E1 +30.868,E3 +209147.720,E4 +0.000} C_DIS
LIN {X -189.654,Y +1120.856,Z +0.000,A -20.000,E1 +39.018,E3 +209169.734,E4 +0.000} C_DIS
LIN {X -195.246,Y +1107.046,Z +0.000,A -20.000,E1 +44.515,E3 +209187.636,E4 +0.000} C_DIS
LIN {X -198.051,Y +1092.368,Z +0.000,A -20.000,E1 +47.947,E3 +209204.162,E4 +0.000} C_DIS
LIN {X -198.143,Y +1081.370,Z +0.000,A -19.806,E1 +49.153,E3 +209216.023,E4 +0.000} C_DIS
